(* IEC 61131-3 sources: Elmo_Master/test/Reports_Lasal/C78_20260806_preemption_cleanup_split (part 3) *)

		groupHeaderPublished := FALSE;
		if restorePreempt & restoredGroupActive then
			// The compact suffix is shared. Restore the complete captured suffix
			// even when the active Group is disjoint from the selected rollback
			// axes, and keep its shared header invalid until every record is done.
			identityHeaderBase := LMC_OWNER_IDENTITY_GROUP_HEADER_BASE;
			OwnershipIdentityState[identityHeaderBase] := 0;
			_memcpy(ptr1:=#OwnershipIdentityState[0],
				ptr2:=#OwnershipPreemptedIdentityState[0],
				cntr:=LMC_OWNER_IDENTITY_SUFFIX_BYTES);
			_memset(dest:=#OwnershipIdentityState[identityHeaderBase],
				usByte:=0, cntr:=40);
			OwnershipIdentityState[identityHeaderBase + 1] :=
				LMC_OWNER_IDENTITY_VERSION;
			OwnershipIdentityState[identityHeaderBase + 2]$UDINT :=
				restoredGroupIdentitySize;
			OwnershipIdentityState[identityHeaderBase + 3]$UDINT :=
				restoredGroupToken;
			OwnershipIdentityState[identityHeaderBase + 4]$UDINT :=
				restoredGroupGeneration;
			OwnershipIdentityState[identityHeaderBase + 5]$UDINT :=
				restoredGroupMask;
			OwnershipIdentityState[identityHeaderBase + 6]$UDINT :=
				restoredGroupSession;
			OwnershipIdentityState[identityHeaderBase + 7]$UDINT :=
				restoredGroupSequence;
			OwnershipIdentityState[identityHeaderBase + 8]$UDINT :=
				TO_UDINT(restoredGroupCommand) or
				(TO_UDINT(restoredGroupReference) shl 16);
			OwnershipIdentityState[identityHeaderBase + 9]$UDINT :=
				TO_UDINT(LMC_OWNER_KIND_GROUP) or
				(TO_UDINT(LMC_OWNER_RESOURCE_AXIS) shl 8) or
				(TO_UDINT(restoredGroupAdmissionMode) shl 16);
			groupHeaderPublished := TRUE;
		end_if;
		axisIndex := 1;
		while axisIndex <= LMC_OWNER_AXIS_COUNT do
			case axisIndex of
				1: axisBit := 0x00000001;
				2: axisBit := 0x00000002;
				3: axisBit := 0x00000004;
				4: axisBit := 0x00000008;
				5: axisBit := 0x00000010;
				6: axisBit := 0x00000020;
				7: axisBit := 0x00000040;
				8: axisBit := 0x00000080;
				9: axisBit := 0x00000100;
			else
				axisBit := 0;
			end_case;
			if (expectedAxisMask and axisBit) <> 0 then
				recordBase := LMC_OWNER_GLOBAL_SLOTS +
					((axisIndex - 1) * LMC_OWNER_AXIS_STRIDE);
				clearIndex := (axisIndex - 1) * LMC_OWNER_AXIS_STRIDE;
				observerBase := (axisIndex - 1) *
					LMC_OWNER_OBSERVER_STRIDE;
				identityHeaderBase := LMC_OWNER_IDENTITY_AXIS_HEADER_BASE +
					((axisIndex - 1) *
					 LMC_OWNER_IDENTITY_AXIS_HEADER_STRIDE);
				OwnershipIdentityState[identityHeaderBase] := 0;
				_memset(dest:=#OwnershipIdentityState[identityHeaderBase],
					usByte:=0,
					cntr:=LMC_OWNER_IDENTITY_AXIS_HEADER_STRIDE * 4);
				if restorePreempt then
					_memcpy(ptr1:=#OwnershipState[recordBase],
						ptr2:=#OwnershipPreemptedState[clearIndex],
						cntr:=LMC_OWNER_AXIS_STRIDE * 4);
					_memcpy(ptr1:=#OwnershipObserverState[observerBase],
						ptr2:=#OwnershipPreemptedIdentityState[
						 LMC_OWNER_PREEMPT_OBSERVER_BASE + observerBase],
						cntr:=LMC_OWNER_OBSERVER_STRIDE * 4);
				else
					_memcpy(ptr1:=#OwnershipState[recordBase],
						ptr2:=#OwnershipLeaseState[clearIndex],
						cntr:=LMC_OWNER_AXIS_STRIDE * 4);
					_memset(dest:=#OwnershipObserverState[observerBase],
						usByte:=0, cntr:=LMC_OWNER_OBSERVER_STRIDE * 4);
				end_if;
				if OwnershipState[recordBase + 1] <> LMC_OWNER_STATE_IDLE then
				identitySize := OwnershipState[recordBase + 15]$UDINT;
				identityTailSize := 0;
				if identitySize > LMC_OWNER_IDENTITY_PREFIX_BYTES then
					identityTailSize := identitySize -
						LMC_OWNER_IDENTITY_PREFIX_BYTES;
				end_if;
				identityPackedCommand :=
					TO_UDINT(OwnershipState[recordBase + 3]) or
					(TO_UDINT(OwnershipState[recordBase + 12]) shl 16);
				identityPackedOwner :=
					TO_UDINT(OwnershipState[recordBase + 2]) or
					(TO_UDINT(OwnershipState[recordBase + 13]) shl 8) or
					(TO_UDINT(OwnershipState[recordBase + 14]) shl 16);
				if OwnershipState[recordBase + 2] =
				   LMC_OWNER_KIND_GROUP then
					if groupHeaderPublished = FALSE then
						identityHeaderBase :=
							LMC_OWNER_IDENTITY_GROUP_HEADER_BASE;
						OwnershipIdentityState[identityHeaderBase] := 0;
						if restorePreempt then
							_memcpy(ptr1:=#OwnershipIdentityState[0],
								ptr2:=#OwnershipPreemptedIdentityState[0],
								cntr:=LMC_OWNER_IDENTITY_SUFFIX_BYTES);
							_memset(dest:=#OwnershipIdentityState[
								identityHeaderBase], usByte:=0, cntr:=40);
							OwnershipIdentityState[identityHeaderBase + 1] :=
								LMC_OWNER_IDENTITY_VERSION;
							OwnershipIdentityState[identityHeaderBase + 2]$UDINT :=
								identitySize;
							OwnershipIdentityState[identityHeaderBase + 3]$UDINT :=
								OwnershipState[recordBase + 4]$UDINT;
							OwnershipIdentityState[identityHeaderBase + 4]$UDINT :=
								OwnershipState[recordBase + 5]$UDINT;
							OwnershipIdentityState[identityHeaderBase + 5]$UDINT :=
								OwnershipState[recordBase + 11]$UDINT;
							OwnershipIdentityState[identityHeaderBase + 6]$UDINT :=
								OwnershipState[recordBase + 6]$UDINT;
							OwnershipIdentityState[identityHeaderBase + 7]$UDINT :=
								OwnershipState[recordBase + 7]$UDINT;
							OwnershipIdentityState[identityHeaderBase + 8]$UDINT :=
								identityPackedCommand;
							OwnershipIdentityState[identityHeaderBase + 9]$UDINT :=
								identityPackedOwner;
						else
							_memcpy(ptr1:=#OwnershipIdentityState[0],
								ptr2:=#OwnershipLeaseIdentityState[0],
								cntr:=LMC_OWNER_IDENTITY_SUFFIX_BYTES);
							_memset(dest:=#OwnershipIdentityState[
								identityHeaderBase], usByte:=0, cntr:=40);
							clearIndex := 1;
							while clearIndex <= 9 do
								OwnershipIdentityState[
									identityHeaderBase + clearIndex] :=
									OwnershipLeaseIdentityState[
									 LMC_OWNER_LEASE_IDENTITY_HEADER_BASE + clearIndex];
								clearIndex += 1;
							end_while;
						end_if;
						groupHeaderPublished := TRUE;
					end_if;
				else
					identityTailOffset :=
						TO_UDINT(OwnershipState[recordBase + 12] - 1) * 8;
					if restorePreempt then
						if identityTailSize > 0 then
							_memset(dest:=#OwnershipIdentityState[
								TO_DINT(identityTailOffset / 4)], usByte:=0,
								cntr:=identityTailSize);
							_memcpy(ptr1:=#OwnershipIdentityState[
								TO_DINT(identityTailOffset / 4)],
								ptr2:=#OwnershipPreemptedIdentityState[
								 TO_DINT(identityTailOffset / 4)],
								cntr:=identityTailSize);
						end_if;
					end_if;
					identityHeaderBase := LMC_OWNER_IDENTITY_AXIS_HEADER_BASE +
						((axisIndex - 1) *
						 LMC_OWNER_IDENTITY_AXIS_HEADER_STRIDE);
					OwnershipIdentityState[identityHeaderBase + 1] :=
						LMC_OWNER_IDENTITY_VERSION;
					OwnershipIdentityState[identityHeaderBase + 2]$UDINT :=
						identitySize;
					OwnershipIdentityState[identityHeaderBase + 3]$UDINT :=
						OwnershipState[recordBase + 4]$UDINT;
					OwnershipIdentityState[identityHeaderBase + 4]$UDINT :=
						OwnershipState[recordBase + 5]$UDINT;
					OwnershipIdentityState[identityHeaderBase + 5]$UDINT :=
						OwnershipState[recordBase + 11]$UDINT;
					OwnershipIdentityState[identityHeaderBase + 6]$UDINT :=
						OwnershipState[recordBase + 6]$UDINT;
					OwnershipIdentityState[identityHeaderBase + 7]$UDINT :=
						OwnershipState[recordBase + 7]$UDINT;
					OwnershipIdentityState[identityHeaderBase + 8]$UDINT :=
						identityPackedCommand;
					OwnershipIdentityState[identityHeaderBase + 9]$UDINT :=
						identityPackedOwner;
					OwnershipIdentityState[identityHeaderBase + 10]$UDINT :=
						identityTailOffset;
					OwnershipIdentityState[identityHeaderBase + 11]$UDINT :=
						identityTailSize;
					OwnershipIdentityState[identityHeaderBase]$UDINT :=
						LMC_OWNER_IDENTITY_AXIS_MAGIC + TO_UDINT(axisIndex);
				end_if;
				end_if;
			end_if;
			axisIndex += 1;
		end_while;
		if groupHeaderPublished then
			OwnershipIdentityState[
				LMC_OWNER_IDENTITY_GROUP_HEADER_BASE]$UDINT :=
				LMC_OWNER_IDENTITY_GROUP_MAGIC;
		end_if;

		if restorePreempt then
			OwnershipPreemptedIdentityState[
				LMC_OWNER_PREEMPT_HEADER_BASE] := 0;
			_memset(dest:=#OwnershipPreemptedState[0], usByte:=0,
				cntr:=sizeof(OwnershipPreemptedState));
			_memset(dest:=#OwnershipPreemptedIdentityState[0], usByte:=0,
				cntr:=sizeof(OwnershipPreemptedIdentityState));
			if restoredGroupActive = FALSE then
				OwnershipLeaseIdentityState[
					LMC_OWNER_LEASE_IDENTITY_HEADER_BASE] := 0;
				_memset(dest:=#OwnershipLeaseState[0], usByte:=0,
					cntr:=sizeof(OwnershipLeaseState));
				_memset(dest:=#OwnershipLeaseIdentityState[0], usByte:=0,
					cntr:=sizeof(OwnershipLeaseIdentityState));
			end_if;
		else
			OwnershipLeaseIdentityState[
				LMC_OWNER_LEASE_IDENTITY_HEADER_BASE] := 0;
			_memset(dest:=#OwnershipLeaseState[0], usByte:=0,
				cntr:=sizeof(OwnershipLeaseState));
			_memset(dest:=#OwnershipLeaseIdentityState[0], usByte:=0,
				cntr:=sizeof(OwnershipLeaseIdentityState));
		end_if;
	elsif Reason = 0 then
		axisIndex := 1;
		while axisIndex <= LMC_OWNER_AXIS_COUNT do
			case axisIndex of
				1: axisBit := 0x00000001;
				2: axisBit := 0x00000002;
				3: axisBit := 0x00000004;
				4: axisBit := 0x00000008;
				5: axisBit := 0x00000010;
				6: axisBit := 0x00000020;
				7: axisBit := 0x00000040;
				8: axisBit := 0x00000080;
				9: axisBit := 0x00000100;
			else
				axisBit := 0;
			end_case;
			if (expectedAxisMask and axisBit) <> 0 then
				recordBase := LMC_OWNER_GLOBAL_SLOTS +
					((axisIndex - 1) * LMC_OWNER_AXIS_STRIDE);
				observerBase := (axisIndex - 1) *
					LMC_OWNER_OBSERVER_STRIDE;
				identityHeaderBase := LMC_OWNER_IDENTITY_AXIS_HEADER_BASE +
					((axisIndex - 1) *
					 LMC_OWNER_IDENTITY_AXIS_HEADER_STRIDE);
				OwnershipIdentityState[identityHeaderBase] := 0;
				_memset(dest:=#OwnershipState[recordBase], usByte:=0,
					cntr:=LMC_OWNER_AXIS_STRIDE * 4);
				OwnershipState[recordBase] := axisIndex;
				OwnershipState[recordBase + 35]$UDINT :=
					LMC_OWNER_AXIS_RECORD_MAGIC + TO_UDINT(axisIndex);
				_memset(dest:=#OwnershipObserverState[observerBase], usByte:=0,
					cntr:=LMC_OWNER_OBSERVER_STRIDE * 4);
			end_if;
			axisIndex += 1;
		end_while;
		if expectedOwnerKind = LMC_OWNER_KIND_GROUP then
			OwnershipIdentityState[
				LMC_OWNER_IDENTITY_GROUP_HEADER_BASE] := 0;
			if expectedAdmissionMode <> LMC_OWNER_ADMISSION_SAFETY then
				_memset(dest:=#OwnershipIdentityState[0], usByte:=0,
					cntr:=LMC_OWNER_IDENTITY_SUFFIX_BYTES);
			end_if;
			_memset(dest:=#OwnershipIdentityState[
				LMC_OWNER_IDENTITY_GROUP_HEADER_BASE], usByte:=0, cntr:=40);
		elsif expectedIdentitySize > LMC_OWNER_IDENTITY_PREFIX_BYTES then
			identityTailSize := expectedIdentitySize -
				LMC_OWNER_IDENTITY_PREFIX_BYTES;
			identityTailOffset := TO_UDINT(expectedReference - 1) * 8;
			_memset(dest:=#OwnershipIdentityState[
				TO_DINT(identityTailOffset / 4)], usByte:=0,
				cntr:=identityTailSize);
		end_if;
	else
		axisIndex := 1;
		while axisIndex <= LMC_OWNER_AXIS_COUNT do
			case axisIndex of
				1: axisBit := 0x00000001;
				2: axisBit := 0x00000002;
				3: axisBit := 0x00000004;
				4: axisBit := 0x00000008;
				5: axisBit := 0x00000010;
				6: axisBit := 0x00000020;
				7: axisBit := 0x00000040;
				8: axisBit := 0x00000080;
				9: axisBit := 0x00000100;
			else
				axisBit := 0;
			end_case;
			if (expectedAxisMask and axisBit) <> 0 then
				recordBase := LMC_OWNER_GLOBAL_SLOTS +
					((axisIndex - 1) * LMC_OWNER_AXIS_STRIDE);
				OwnershipState[recordBase + 1] :=
					LMC_OWNER_STATE_QUARANTINED;
				OwnershipState[recordBase + 32] :=
					LMC_OWNER_REPORT_QUARANTINE;
				OwnershipState[recordBase + 33] := Reason;
			end_if;
			axisIndex += 1;
		end_while;
	end_if;
	if (Reason = 0) &
	   (OwnershipState[7]$UDINT = AdmissionToken) &
	   (OwnershipState[8]$UDINT = OwnerGeneration) then
		OwnershipState[7] := 0;
		OwnershipState[8] := 0;
		OwnershipState[9] := 0;
	end_if;
	if (Reason = 0) &
	   (OwnershipState[10]$UDINT = AdmissionToken) &
	   (OwnershipState[11]$UDINT = OwnerGeneration) then
		OwnershipState[10] := 0;
		OwnershipState[11] := 0;
		OwnershipState[12] := 0;
	end_if;
	if (Reason = 0) &
	   (OwnershipState[13]$UDINT = AdmissionToken) &
	   (OwnershipState[14]$UDINT = OwnerGeneration) then
		OwnershipState[13] := 0;
		OwnershipState[14] := 0;
		OwnershipState[15] := 0;
	end_if;
	Result := 0;

END_FUNCTION

FUNCTION GLOBAL LMCControlCommandService::PublishAxisOwnership
	VAR_INPUT
		AxisMask : UDINT;
		AdmissionToken : UDINT;
		OwnerGeneration : UDINT;
		ReportKind : UINT;
		ReportValue0 : UDINT;
		ReportValue1 : UDINT;
		ObservationCycle : UDINT;
	END_VAR
	VAR_OUTPUT
		Result : DINT;
	END_VAR
	VAR
		axisIndex : DINT;
		axisBit : UDINT;
		recordBase : DINT;
		firstRecordBase : DINT;
		leaseRecordBase : DINT;
		leaseFirstRecordBase : DINT;
		preemptRecordBase : DINT;
		probeRecordBase : DINT;
		probeAxisIndex : DINT;
		probeAxisBit : UDINT;
		observerBase : DINT;
		observerIndex : DINT;
		identityIndex : DINT;
		clearIndex : DINT;
		identityHeaderBase : DINT;
		identityCompareResult : UDINT;
		expectedResourceKind : DINT;
		expectedOwnerKind : DINT;
		expectedCommandId : DINT;
		expectedAdmissionMode : DINT;
		expectedReference : DINT;
		expectedSession : UDINT;
		expectedSequence : UDINT;
		observerFlags : UDINT;
		preemptFlags : UDINT;
		cleanupRequiredMask : UDINT;
		cleanupCompleteMask : UDINT;
		identitySize : UDINT;
		identityPrefixSize : UDINT;
		identityTailSize : UDINT;
		identityTailOffset : UDINT;
		identityPackedCommand : UDINT;
		identityPackedOwner : UDINT;
		preemptToken : UDINT;
		preemptGeneration : UDINT;
		preemptSession : UDINT;
		preemptSequence : UDINT;
		preemptMask : UDINT;
		preemptIdentitySize : UDINT;
		preemptState : DINT;
		preemptOwnerKind : DINT;
		preemptResourceKind : DINT;
		preemptCommand : DINT;
		preemptReference : DINT;
		preemptAdmission : DINT;
		replacementRecordBase : DINT;
		replacementHeaderBase : DINT;
		singletonToken : UDINT;
		singletonGeneration : UDINT;
		singletonMask : UDINT;
		replacementIdentitySize : UDINT;
		replacementTailSize : UDINT;
		replacementTailOffset : UDINT;
		replacementPackedCommand : UDINT;
		replacementPackedOwner : UDINT;
		resourceValid : BOOL;
		selectedFound : BOOL;
		identityShapeValid : BOOL;
		retainGroupLease : BOOL;
		forceQuarantine : BOOL;
		preemptRootValid : BOOL;
		cleanupReady : BOOL;
		restoreLease : BOOL;
		leaseValid : BOOL;
		retainLeaseValid : BOOL;
		preemptBankValid : BOOL;
		preemptSpecialValid : BOOL;
		replacementFound : BOOL;
		replacementValid : BOOL;
		replacementStateValid : BOOL;
		preemptLmcFound : BOOL;
		preemptDs402Found : BOOL;
		preemptEncoderFound : BOOL;
		destroyBanks : BOOL;
		clearOwner : BOOL;
		groupHeaderPublished : BOOL;
		homeReceiptExact : BOOL;
		homeReceiptCallMatches : BOOL;
		homeReceiptTerminalComplete : BOOL;
		homeReceiptAxisMaskValid : BOOL;
		homeReceiptIdentityPre : BOOL;
		homeReceiptIdentityPost : BOOL;
		homeReceiptObserverPre : BOOL;
		homeReceiptObserverPost : BOOL;
		homeReceiptRecordPre : BOOL;
		homeReceiptRecordBodyPost : BOOL;
		homeReceiptRecordPost : BOOL;
		homeReceiptSingletonPre : BOOL;
		homeReceiptSingletonPost : BOOL;
		homeReceiptSurfaceValid : BOOL;
		homeReceiptPhase : DINT;
		homeReceiptIndex : DINT;
		rebaseUpdateResult : DINT;
	END_VAR

	Result := -1;
	if (AxisMask = 0) | (AxisMask > LMC_OWNER_ROBOT_AXIS_MASK) |
	   (AdmissionToken = 0) | (OwnerGeneration = 0) |
	   (ReportKind < LMC_OWNER_REPORT_DISPATCH) |
	   (ReportKind > LMC_OWNER_REPORT_SAFETY_PREEMPT) then
		RETURN;
	end_if;
	if ZeroHomeState[60]$UDINT = LMC_HOME_OWNER_RECEIPT_MAGIC then
		homeReceiptCallMatches :=
			(ZeroHomeState[34]$UDINT = AdmissionToken) &
			(ZeroHomeState[35]$UDINT = OwnerGeneration) &
			(ZeroHomeState[38]$UDINT = AxisMask) &
			(ZeroHomeState[58] = TO_DINT(ReportKind)) &
			(ZeroHomeState[57]$UDINT = ReportValue0) &
			(ZeroHomeState[31]$UDINT = ReportValue1) &
			(ZeroHomeState[46]$UDINT = ObservationCycle);
		homeReceiptTerminalComplete :=
			(ZeroHomeState[51]$UDINT = LMC_HOME_RECORD_MAGIC) &
			(ZeroHomeState[33]$UDINT <> 0) &
			(ZeroHomeState[63]$UDINT = ZeroHomeState[33]$UDINT) &
			(ZeroHomeState[62] = 0) &
			(ZeroHomeState[61] = LMC_HOME_OWNER_RECEIPT_COMPLETE) &
			(ZeroHomeState[59] = 0) &
			(ZeroHomeState[39] = LMC_HOME_ENGINE_TERMINAL) &
			(ZeroHomeState[0] >= LMC_HOME_RECORD_SUCCEEDED) &
			(ZeroHomeState[0] <= LMC_HOME_RECORD_ABORTED) &
			(ZeroHomeState[57] = ZeroHomeState[0]) &
			(ZeroHomeState[47] = 1) &
			((ZeroHomeState[56]$UDINT and
			  LMC_HOME_FLAG_OWNER_FINALIZE_ACCEPTED) <> 0) &
			((ZeroHomeState[56]$UDINT and
			  LMC_HOME_FLAG_TERMINAL_PUBLISHED) <> 0) &
			((ZeroHomeState[56]$UDINT and
			  LMC_HOME_FLAG_PREEMPTION_CLEANUP) = 0) &
			(((ZeroHomeState[0] = LMC_HOME_RECORD_SUCCEEDED) &
			  (ZeroHomeState[58] = LMC_OWNER_REPORT_TERMINAL_SUCCESS)) |
			 (((ZeroHomeState[0] = LMC_HOME_RECORD_FAILED) |
			   (ZeroHomeState[0] = LMC_HOME_RECORD_ABORTED)) &
			  (ZeroHomeState[58] =
			   LMC_OWNER_REPORT_TERMINAL_SAFE_FAILURE)));
		if homeReceiptCallMatches then
		homeReceiptPhase := ZeroHomeState[61];
		homeReceiptAxisMaskValid := FALSE;
		case ZeroHomeState[9] of
			1: homeReceiptAxisMaskValid := AxisMask = 0x00000001;
			2: homeReceiptAxisMaskValid := AxisMask = 0x00000002;
			3: homeReceiptAxisMaskValid := AxisMask = 0x00000004;
			4: homeReceiptAxisMaskValid := AxisMask = 0x00000008;
		else
		end_case;
		homeReceiptExact :=
			homeReceiptAxisMaskValid &
			(ZeroHomeState[51]$UDINT = LMC_HOME_RECORD_MAGIC) &
			(ZeroHomeState[33]$UDINT <> 0) &
			(ZeroHomeState[63]$UDINT = ZeroHomeState[33]$UDINT) &
			(ZeroHomeState[62] = 0) &
			(ZeroHomeState[34]$UDINT = AdmissionToken) &
			(ZeroHomeState[35]$UDINT = OwnerGeneration) &
			(ZeroHomeState[38]$UDINT = AxisMask) &
			(ZeroHomeState[58] = TO_DINT(ReportKind)) &
			(ZeroHomeState[57]$UDINT = ReportValue0) &
			(ZeroHomeState[31]$UDINT = ReportValue1) &
			(ZeroHomeState[46]$UDINT = ObservationCycle) &
			(ZeroHomeState[59] = 0) &
			((ZeroHomeState[39] = LMC_HOME_ENGINE_FINALIZE) |
			 (ZeroHomeState[39] = LMC_HOME_ENGINE_TERMINAL)) &
			((ZeroHomeState[56]$UDINT and
			  LMC_HOME_FLAG_OWNER_FINALIZE_INTENT) <> 0) &
			((ZeroHomeState[56]$UDINT and
			  LMC_HOME_FLAG_PREEMPTION_CLEANUP) = 0) &
			((ReportKind = LMC_OWNER_REPORT_TERMINAL_SUCCESS) |
			 (ReportKind = LMC_OWNER_REPORT_TERMINAL_SAFE_FAILURE)) &
			(homeReceiptPhase >= LMC_HOME_OWNER_RECEIPT_PREPARED) &
			(homeReceiptPhase <= LMC_HOME_OWNER_RECEIPT_COMPLETE);
		if homeReceiptExact = FALSE then
			OwnershipState[24] := 1;
			Result := -3;
			RETURN;
		end_if;

		axisIndex := ZeroHomeState[9];
		recordBase := LMC_OWNER_GLOBAL_SLOTS +
			((axisIndex - 1) * LMC_OWNER_AXIS_STRIDE);
		observerBase := (axisIndex - 1) * LMC_OWNER_OBSERVER_STRIDE;
		identityHeaderBase := LMC_OWNER_IDENTITY_AXIS_HEADER_BASE +
			((axisIndex - 1) * LMC_OWNER_IDENTITY_AXIS_HEADER_STRIDE);
		identityPackedCommand := TO_UDINT(0x7D13) or
			(TO_UDINT(axisIndex) shl 16);
		identityPackedOwner := TO_UDINT(LMC_OWNER_KIND_LMC_HOME) or
			(TO_UDINT(LMC_OWNER_RESOURCE_LMC_HOME_ENGINE) shl 8) or
			(TO_UDINT(LMC_OWNER_ADMISSION_LIFECYCLE) shl 16);
		identitySize := OwnershipState[recordBase + 15]$UDINT;
		identityTailOffset := TO_UDINT(axisIndex - 1) * 8;
		identityTailSize := 0;
		if identitySize > LMC_OWNER_IDENTITY_PREFIX_BYTES then
			identityTailSize := identitySize - LMC_OWNER_IDENTITY_PREFIX_BYTES;
		end_if;

		homeReceiptIdentityPre :=
			(OwnershipIdentityState[identityHeaderBase]$UDINT =
			 (LMC_OWNER_IDENTITY_AXIS_MAGIC + TO_UDINT(axisIndex))) &
			(OwnershipIdentityState[identityHeaderBase + 1] =
			 LMC_OWNER_IDENTITY_VERSION) &
			(OwnershipIdentityState[identityHeaderBase + 2]$UDINT = 56) &
			(OwnershipIdentityState[identityHeaderBase + 3]$UDINT =
			 AdmissionToken) &
			(OwnershipIdentityState[identityHeaderBase + 4]$UDINT =
			 OwnerGeneration) &
			(OwnershipIdentityState[identityHeaderBase + 5]$UDINT = AxisMask) &
			(OwnershipIdentityState[identityHeaderBase + 6]$UDINT =
			 ZeroHomeState[36]$UDINT) &
			(OwnershipIdentityState[identityHeaderBase + 7]$UDINT =
			 ZeroHomeState[37]$UDINT) &
			(OwnershipIdentityState[identityHeaderBase + 8]$UDINT =
			 identityPackedCommand) &
			(OwnershipIdentityState[identityHeaderBase + 9]$UDINT =
			 identityPackedOwner) &
			(OwnershipIdentityState[identityHeaderBase + 10]$UDINT =
			 identityTailOffset) &
			(OwnershipIdentityState[identityHeaderBase + 11]$UDINT = 0) &
			(identitySize = 56) & (identityTailSize = 0);
		homeReceiptIdentityPost := TRUE;
		homeReceiptIndex := 0;
		while homeReceiptIndex < LMC_OWNER_IDENTITY_AXIS_HEADER_STRIDE do
			if OwnershipIdentityState[identityHeaderBase + homeReceiptIndex] <> 0 then
				homeReceiptIdentityPost := FALSE;
			end_if;
			homeReceiptIndex += 1;
		end_while;

		homeReceiptObserverPre :=
			(OwnershipObserverState[observerBase]$UDINT =
			 (LMC_OWNER_OBSERVER_MAGIC + TO_UDINT(axisIndex))) &
			(OwnershipObserverState[observerBase + 1]$UDINT = AdmissionToken) &
			(OwnershipObserverState[observerBase + 2]$UDINT = OwnerGeneration) &
			((OwnershipObserverState[observerBase + 5]$UDINT and
			  LMC_OWNER_OBSERVER_EVIDENCE_CLEAR_MASK) = 0) &
			(OwnershipObserverState[observerBase + 9] = 0) &
			(OwnershipObserverState[observerBase + 10] = 0) &
			(OwnershipObserverState[observerBase + 11] = 0);
		homeReceiptObserverPost := TRUE;
		homeReceiptIndex := 0;
		while homeReceiptIndex < LMC_OWNER_OBSERVER_STRIDE do
			if OwnershipObserverState[observerBase + homeReceiptIndex] <> 0 then
				homeReceiptObserverPost := FALSE;
			end_if;
			homeReceiptIndex += 1;
		end_while;

		homeReceiptRecordPre :=
			(OwnershipState[recordBase] = axisIndex) &
			(OwnershipState[recordBase + 1] = LMC_OWNER_STATE_LMC_HOME_ACTIVE) &
			(OwnershipState[recordBase + 2] = LMC_OWNER_KIND_LMC_HOME) &
			(OwnershipState[recordBase + 3] = 0x7D13) &
			(OwnershipState[recordBase + 4]$UDINT = AdmissionToken) &
			(OwnershipState[recordBase + 5]$UDINT = OwnerGeneration) &
			(OwnershipState[recordBase + 6]$UDINT = ZeroHomeState[36]$UDINT) &
			(OwnershipState[recordBase + 7]$UDINT = ZeroHomeState[37]$UDINT) &
			(OwnershipState[recordBase + 8]$UDINT <> 0) &
			(OwnershipState[recordBase + 9]$UDINT <> 0) &
			(OwnershipState[recordBase + 10] = 0) &
			(OwnershipState[recordBase + 11]$UDINT = AxisMask) &
			(OwnershipState[recordBase + 12] = axisIndex) &
			(OwnershipState[recordBase + 13] =
			 LMC_OWNER_RESOURCE_LMC_HOME_ENGINE) &
			(OwnershipState[recordBase + 14] =
			 LMC_OWNER_ADMISSION_LIFECYCLE) &
			(OwnershipState[recordBase + 15]$UDINT = 56) &
			(OwnershipState[recordBase + 16]$UDINT = 1) &
			(OwnershipState[recordBase + 17]$UDINT = ZeroHomeState[4]$UDINT) &
			(OwnershipState[recordBase + 18]$UDINT = ZeroHomeState[1]$UDINT) &
			(OwnershipState[recordBase + 19]$UDINT = ZeroHomeState[2]$UDINT) &
			(OwnershipState[recordBase + 20]$UDINT = ZeroHomeState[3]$UDINT) &
			(OwnershipState[recordBase + 21]$UDINT = ZeroHomeState[5]$UDINT) &
			(OwnershipState[recordBase + 22]$UDINT = ZeroHomeState[6]$UDINT) &
			(OwnershipState[recordBase + 23]$UDINT = ZeroHomeState[7]$UDINT) &
			(OwnershipState[recordBase + 24]$UDINT = ZeroHomeState[8]$UDINT) &
			(OwnershipState[recordBase + 25]$UDINT = 1) &
			(OwnershipState[recordBase + 26] = ZeroHomeState[11]) &
			(OwnershipState[recordBase + 27] = ZeroHomeState[12]) &
			(OwnershipState[recordBase + 28]$UDINT = ZeroHomeState[13]$UDINT) &
			(OwnershipState[recordBase + 29]$UDINT = 0x454D4F48) &
			(OwnershipState[recordBase + 30] = 0) &
			(OwnershipState[recordBase + 31] = 0) &
			(OwnershipState[recordBase + 32] = 0) &
			(OwnershipState[recordBase + 33] = 0) &
			(OwnershipState[recordBase + 34] = 0) &
			(OwnershipState[recordBase + 35]$UDINT =
			 (LMC_OWNER_AXIS_RECORD_MAGIC + TO_UDINT(axisIndex)));
		homeReceiptRecordBodyPost := OwnershipState[recordBase] = axisIndex;
		homeReceiptIndex := 1;
		while homeReceiptIndex <= 34 do
			if OwnershipState[recordBase + homeReceiptIndex] <> 0 then
				homeReceiptRecordBodyPost := FALSE;
			end_if;
			homeReceiptIndex += 1;
		end_while;
		homeReceiptRecordPost := homeReceiptRecordBodyPost &
			(OwnershipState[recordBase + 35]$UDINT =
			 (LMC_OWNER_AXIS_RECORD_MAGIC + TO_UDINT(axisIndex)));
		homeReceiptSingletonPre :=
			(OwnershipState[7]$UDINT = AdmissionToken) &
			(OwnershipState[8]$UDINT = OwnerGeneration) &
			(OwnershipState[9]$UDINT = AxisMask);
		homeReceiptSingletonPost :=
			(OwnershipState[7]$UDINT = 0) &
			(OwnershipState[8]$UDINT = 0) &
			(OwnershipState[9]$UDINT = 0);

		homeReceiptSurfaceValid := FALSE;
		case homeReceiptPhase of
			LMC_HOME_OWNER_RECEIPT_PREPARED:
				homeReceiptSurfaceValid := homeReceiptIdentityPre &
					homeReceiptObserverPre & homeReceiptRecordPre &
					homeReceiptSingletonPre;
			LMC_HOME_OWNER_RECEIPT_CLEAR_IDENTITY:
				homeReceiptSurfaceValid :=
					(homeReceiptIdentityPre | homeReceiptIdentityPost |
					 (OwnershipIdentityState[identityHeaderBase] = 0)) &
					homeReceiptObserverPre & homeReceiptRecordPre &
					homeReceiptSingletonPre;
			LMC_HOME_OWNER_RECEIPT_CLEAR_OBSERVER:
				homeReceiptSurfaceValid := homeReceiptIdentityPost &
					(homeReceiptObserverPre | homeReceiptObserverPost |
					 (OwnershipObserverState[observerBase] = 0)) &
					homeReceiptRecordPre & homeReceiptSingletonPre;
			LMC_HOME_OWNER_RECEIPT_CLEAR_SINGLETON:
				homeReceiptSurfaceValid := homeReceiptIdentityPost &
					homeReceiptObserverPost & homeReceiptRecordPre &
					(homeReceiptSingletonPre |
					 ((OwnershipState[7]$UDINT = 0) &
					  (OwnershipState[8]$UDINT = OwnerGeneration) &
					  (OwnershipState[9]$UDINT = AxisMask)) |
					 ((OwnershipState[7]$UDINT = 0) &
					  (OwnershipState[8]$UDINT = 0) &
					  (OwnershipState[9]$UDINT = AxisMask)) |
					 homeReceiptSingletonPost);
			LMC_HOME_OWNER_RECEIPT_CLEAR_RECORD:
				homeReceiptSurfaceValid := homeReceiptIdentityPost &
					homeReceiptObserverPost & homeReceiptSingletonPost &
					(homeReceiptRecordPre |
					 (OwnershipState[recordBase + 35] = 0));
			LMC_HOME_OWNER_RECEIPT_COMPLETE:
				homeReceiptSurfaceValid := homeReceiptIdentityPost &
					homeReceiptObserverPost & homeReceiptSingletonPost &
					(homeReceiptRecordPost |
					 (homeReceiptRecordBodyPost &
					  (OwnershipState[recordBase + 35] = 0)));
		else
		end_case;
		if homeReceiptSurfaceValid = FALSE then
			OwnershipState[24] := 1;
			Result := -3;
			RETURN;
		end_if;
		if (ZeroHomeState[56]$UDINT and
		   LMC_HOME_FLAG_OWNER_FINALIZE_ACCEPTED) = 0 then
			if homeReceiptPhase <> LMC_HOME_OWNER_RECEIPT_PREPARED then
				OwnershipState[24] := 1;
				Result := -3;
				RETURN;
			end_if;
			Result := 0;
			RETURN;
		end_if;

		// The axis-record magic is committed last. Each phase is stored before its
		// mutation, so the exact receipt can resume a partial cleanup fail-closed.
		if homeReceiptPhase <= LMC_HOME_OWNER_RECEIPT_CLEAR_IDENTITY then
			ZeroHomeState[61] := LMC_HOME_OWNER_RECEIPT_CLEAR_IDENTITY;
			OwnershipIdentityState[identityHeaderBase] := 0;
			_memset(dest:=#OwnershipIdentityState[identityHeaderBase],
				usByte:=0, cntr:=LMC_OWNER_IDENTITY_AXIS_HEADER_STRIDE * 4);
		end_if;
		if homeReceiptPhase <= LMC_HOME_OWNER_RECEIPT_CLEAR_OBSERVER then
			ZeroHomeState[61] := LMC_HOME_OWNER_RECEIPT_CLEAR_OBSERVER;
			OwnershipObserverState[observerBase] := 0;
			_memset(dest:=#OwnershipObserverState[observerBase],
				usByte:=0, cntr:=LMC_OWNER_OBSERVER_STRIDE * 4);
		end_if;
		if homeReceiptPhase <= LMC_HOME_OWNER_RECEIPT_CLEAR_SINGLETON then
			ZeroHomeState[61] := LMC_HOME_OWNER_RECEIPT_CLEAR_SINGLETON;
			OwnershipState[7] := 0;
			OwnershipState[8] := 0;
			OwnershipState[9] := 0;
		end_if;
		if homeReceiptPhase <= LMC_HOME_OWNER_RECEIPT_CLEAR_RECORD then
			ZeroHomeState[61] := LMC_HOME_OWNER_RECEIPT_CLEAR_RECORD;
			OwnershipState[recordBase + 35] := 0;
			_memset(dest:=#OwnershipState[recordBase], usByte:=0,
				cntr:=LMC_OWNER_AXIS_STRIDE * 4);
			OwnershipState[recordBase] := axisIndex;
			ZeroHomeState[61] := LMC_HOME_OWNER_RECEIPT_COMPLETE;
			OwnershipState[recordBase + 35]$UDINT :=
				LMC_OWNER_AXIS_RECORD_MAGIC + TO_UDINT(axisIndex);
		elsif (homeReceiptPhase = LMC_HOME_OWNER_RECEIPT_COMPLETE) &
		      homeReceiptRecordBodyPost &
		      (OwnershipState[recordBase + 35] = 0) then
			OwnershipState[recordBase + 35]$UDINT :=
				LMC_OWNER_AXIS_RECORD_MAGIC + TO_UDINT(axisIndex);
		end_if;
		if (ZeroHomeState[61] <> LMC_HOME_OWNER_RECEIPT_COMPLETE) |
		   (OwnershipState[recordBase + 35]$UDINT <>
		    (LMC_OWNER_AXIS_RECORD_MAGIC + TO_UDINT(axisIndex))) then
			OwnershipState[24] := 1;
			Result := -3;
			RETURN;
		end_if;
		// Clear only after exact successful Home and durable owner cleanup. The
		// caller has not published ZeroHomeState[0] yet, so the receipt-bound
		// terminal tuple is the authoritative success proof at this point.
		if LMC_AXIS_REBASE_BARRIER_ENABLED &
		   (ReportKind = LMC_OWNER_REPORT_TERMINAL_SUCCESS) &
		   (ReportValue0 = LMC_HOME_RECORD_SUCCEEDED) &
		   (ZeroHomeState[57] = LMC_HOME_RECORD_SUCCEEDED) then
			rebaseUpdateResult := UpdateAxisRebaseRequiredState(
				SetAxisMask:=0, ClearAxisMask:=AxisMask);
			if rebaseUpdateResult <> 0 then
				Result := rebaseUpdateResult;
				RETURN;
			end_if;
		end_if;
		Result := 1;
		RETURN;
		elsif homeReceiptTerminalComplete = FALSE then
			OwnershipState[24] := 1;
			Result := -3;
			RETURN;
		end_if;
	end_if;
	expectedResourceKind := 0;
	expectedOwnerKind := 0;
	expectedCommandId := 0;
	expectedAdmissionMode := 0;
	expectedReference := 0;
	expectedSession := 0;
	expectedSequence := 0;
	identitySize := 0;
	firstRecordBase := -1;
	selectedFound := FALSE;
	axisIndex := 1;
	while axisIndex <= LMC_OWNER_AXIS_COUNT do
		case axisIndex of
			1: axisBit := 0x00000001;
			2: axisBit := 0x00000002;
			3: axisBit := 0x00000004;
			4: axisBit := 0x00000008;
			5: axisBit := 0x00000010;
			6: axisBit := 0x00000020;
			7: axisBit := 0x00000040;
			8: axisBit := 0x00000080;
			9: axisBit := 0x00000100;
		else
			axisBit := 0;
		end_case;
		recordBase := LMC_OWNER_GLOBAL_SLOTS +
			((axisIndex - 1) * LMC_OWNER_AXIS_STRIDE);
		if (AxisMask and axisBit) <> 0 then
			if selectedFound = FALSE then
				expectedResourceKind := OwnershipState[recordBase + 13];
				expectedOwnerKind := OwnershipState[recordBase + 2];
				expectedCommandId := OwnershipState[recordBase + 3];
				expectedAdmissionMode := OwnershipState[recordBase + 14];
				expectedReference := OwnershipState[recordBase + 12];
				expectedSession := OwnershipState[recordBase + 6]$UDINT;
				expectedSequence := OwnershipState[recordBase + 7]$UDINT;
				identitySize := OwnershipState[recordBase + 15]$UDINT;
				firstRecordBase := recordBase;
				selectedFound := TRUE;
			end_if;
			if (OwnershipState[recordBase] <> axisIndex) |
			   (OwnershipState[recordBase + 35]$UDINT <>
			    (LMC_OWNER_AXIS_RECORD_MAGIC + TO_UDINT(axisIndex))) |
			   (OwnershipState[recordBase + 4]$UDINT <>
			    AdmissionToken) |
			   (OwnershipState[recordBase + 5]$UDINT <>
			    OwnerGeneration) |
			   (OwnershipState[recordBase + 11]$UDINT <> AxisMask) |
			   (OwnershipState[recordBase + 13] <>
			    expectedResourceKind) |
			   (OwnershipState[recordBase + 2] <> expectedOwnerKind) |
			   (OwnershipState[recordBase + 3] <> expectedCommandId) |
			   (OwnershipState[recordBase + 14] <>
			    expectedAdmissionMode) |
			   (OwnershipState[recordBase + 12] <>
			    expectedReference) |
			   (OwnershipState[recordBase + 6]$UDINT <> expectedSession) |
			   (OwnershipState[recordBase + 7]$UDINT <> expectedSequence) |
			   (OwnershipState[recordBase + 15]$UDINT <> identitySize) then
				Result := -2;
				RETURN;
			elsif (OwnershipState[recordBase + 1] =
			       LMC_OWNER_STATE_QUARANTINED) &
			      (ReportKind <> LMC_OWNER_REPORT_QUARANTINE) then
				Result := -3;
				RETURN;
			end_if;
		elsif (OwnershipState[recordBase + 4]$UDINT = AdmissionToken) |
		      (OwnershipState[recordBase + 5]$UDINT = OwnerGeneration) then
			Result := -2;
			RETURN;
		end_if;
		axisIndex += 1;
	end_while;
	if selectedFound = FALSE then
		Result := -2;
		RETURN;
	end_if;
	identityShapeValid := FALSE;
	if expectedCommandId = 0x2023 then
		identityShapeValid := identitySize = 8;
	elsif expectedCommandId = 0x2024 then
		identityShapeValid := identitySize = 1;
	elsif expectedCommandId = 0x2022 then
		identityShapeValid := identitySize = 16;
	elsif (expectedCommandId = 0x209F) | (expectedCommandId = 0x20A0) then
		identityShapeValid := identitySize = 32;
	elsif expectedCommandId = 0x20A2 then
		identityShapeValid := identitySize = 24;
	elsif (expectedCommandId = 0x2047) | (expectedCommandId = 0x2048) |
	      (expectedCommandId = 0x2049) | (expectedCommandId = 0x204A) |
	      (expectedCommandId = 0x204B) then
		identityShapeValid := identitySize = 1;
	elsif expectedCommandId = 0x2085 then
		identityShapeValid := identitySize = 16;
	elsif expectedCommandId = 0x20A4 then
		identityShapeValid := identitySize = 96;
	elsif expectedCommandId = 0x7D22 then
		identityShapeValid := identitySize = 104;
	elsif expectedCommandId = 0x20E7 then
		identityShapeValid := identitySize = 1320;
	elsif expectedCommandId = 0x7D13 then
		identityShapeValid := identitySize = 56;
	elsif (expectedCommandId = 0x7D15) |
	      (expectedCommandId = 0x7E53) then
		identityShapeValid := identitySize = 72;
	end_if;
	identityPrefixSize := identitySize;
	if identityPrefixSize > LMC_OWNER_IDENTITY_PREFIX_BYTES then
		identityPrefixSize := LMC_OWNER_IDENTITY_PREFIX_BYTES;
	end_if;
	identityTailSize := 0;
	if identitySize > LMC_OWNER_IDENTITY_PREFIX_BYTES then
		identityTailSize := identitySize - LMC_OWNER_IDENTITY_PREFIX_BYTES;
	end_if;
	identityTailOffset := 0;
	if expectedOwnerKind <> LMC_OWNER_KIND_GROUP then
		if (expectedReference < 1) |
		   (expectedReference > LMC_OWNER_AXIS_COUNT) then
			identityShapeValid := FALSE;
		else
			identityTailOffset := TO_UDINT(expectedReference - 1) * 8;
		end_if;
		if identityTailSize > 8 then
			identityShapeValid := FALSE;
		end_if;
	end_if;
	if (identityTailOffset + identityTailSize) >
	   LMC_OWNER_IDENTITY_SUFFIX_BYTES then
		identityShapeValid := FALSE;
	end_if;
	identityPackedCommand := TO_UDINT(expectedCommandId) or
		(TO_UDINT(expectedReference) shl 16);
	identityPackedOwner := TO_UDINT(expectedOwnerKind) or
		(TO_UDINT(expectedResourceKind) shl 8) or
		(TO_UDINT(expectedAdmissionMode) shl 16);
	axisIndex := 1;
	while axisIndex <= LMC_OWNER_AXIS_COUNT do
		case axisIndex of
			1: axisBit := 0x00000001;
			2: axisBit := 0x00000002;
			3: axisBit := 0x00000004;
			4: axisBit := 0x00000008;
			5: axisBit := 0x00000010;
			6: axisBit := 0x00000020;
			7: axisBit := 0x00000040;
			8: axisBit := 0x00000080;
			9: axisBit := 0x00000100;
		else
			axisBit := 0;
		end_case;
		if (AxisMask and axisBit) <> 0 then
			recordBase := LMC_OWNER_GLOBAL_SLOTS +
				((axisIndex - 1) * LMC_OWNER_AXIS_STRIDE);
			if expectedOwnerKind = LMC_OWNER_KIND_GROUP then
				identityHeaderBase := LMC_OWNER_IDENTITY_GROUP_HEADER_BASE;
				if (OwnershipIdentityState[identityHeaderBase]$UDINT <>
				    LMC_OWNER_IDENTITY_GROUP_MAGIC) |
				   (OwnershipIdentityState[identityHeaderBase + 1] <>
				    LMC_OWNER_IDENTITY_VERSION) |
				   (OwnershipIdentityState[identityHeaderBase + 2]$UDINT <>
				    identitySize) |
				   (OwnershipIdentityState[identityHeaderBase + 3]$UDINT <>
				    AdmissionToken) |
				   (OwnershipIdentityState[identityHeaderBase + 4]$UDINT <>
				    OwnerGeneration) |
				   (OwnershipIdentityState[identityHeaderBase + 5]$UDINT <>
				    AxisMask) |
				   (OwnershipIdentityState[identityHeaderBase + 6]$UDINT <>
				    expectedSession) |
				   (OwnershipIdentityState[identityHeaderBase + 7]$UDINT <>
				    expectedSequence) |
				   (OwnershipIdentityState[identityHeaderBase + 8]$UDINT <>
				    identityPackedCommand) |
				   (OwnershipIdentityState[identityHeaderBase + 9]$UDINT <>
				    identityPackedOwner) then
					identityShapeValid := FALSE;
				end_if;
			else
				identityHeaderBase := LMC_OWNER_IDENTITY_AXIS_HEADER_BASE +
					((axisIndex - 1) * LMC_OWNER_IDENTITY_AXIS_HEADER_STRIDE);
				if (OwnershipIdentityState[identityHeaderBase]$UDINT <>
				    (LMC_OWNER_IDENTITY_AXIS_MAGIC + TO_UDINT(axisIndex))) |
				   (OwnershipIdentityState[identityHeaderBase + 1] <>
				    LMC_OWNER_IDENTITY_VERSION) |
				   (OwnershipIdentityState[identityHeaderBase + 2]$UDINT <>
				    identitySize) |
				   (OwnershipIdentityState[identityHeaderBase + 3]$UDINT <>
				    AdmissionToken) |
				   (OwnershipIdentityState[identityHeaderBase + 4]$UDINT <>
				    OwnerGeneration) |
				   (OwnershipIdentityState[identityHeaderBase + 5]$UDINT <>
				    AxisMask) |
				   (OwnershipIdentityState[identityHeaderBase + 6]$UDINT <>
				    expectedSession) |
				   (OwnershipIdentityState[identityHeaderBase + 7]$UDINT <>
				    expectedSequence) |
				   (OwnershipIdentityState[identityHeaderBase + 8]$UDINT <>
				    identityPackedCommand) |
				   (OwnershipIdentityState[identityHeaderBase + 9]$UDINT <>
				    identityPackedOwner) |
				   (OwnershipIdentityState[identityHeaderBase + 10]$UDINT <>
				    identityTailOffset) |
				   (OwnershipIdentityState[identityHeaderBase + 11]$UDINT <>
				    identityTailSize) then
					identityShapeValid := FALSE;
				end_if;
			end_if;
			identityCompareResult := _memcmp(
				ptr1:=#OwnershipState[firstRecordBase + 16],
				ptr2:=#OwnershipState[recordBase + 16],
				cntr:=identityPrefixSize);
			if identityCompareResult <> 0 then
				identityShapeValid := FALSE;
			end_if;
		end_if;
		axisIndex += 1;
	end_while;
	if identityShapeValid = FALSE then
		OwnershipState[24] := 1;
		Result := -3;
		RETURN;
	end_if;
	resourceValid := FALSE;
	case expectedResourceKind of
		LMC_OWNER_RESOURCE_AXIS:
			resourceValid :=
				(OwnershipState[7]$UDINT <> AdmissionToken) &
				(OwnershipState[8]$UDINT <> OwnerGeneration) &
				(OwnershipState[10]$UDINT <> AdmissionToken) &
				(OwnershipState[11]$UDINT <> OwnerGeneration) &
				(OwnershipState[13]$UDINT <> AdmissionToken) &
				(OwnershipState[14]$UDINT <> OwnerGeneration);
		LMC_OWNER_RESOURCE_LMC_HOME_ENGINE:
			resourceValid :=
				(OwnershipState[7]$UDINT = AdmissionToken) &
				(OwnershipState[8]$UDINT = OwnerGeneration) &
				(OwnershipState[9]$UDINT = AxisMask) &
				(OwnershipState[10]$UDINT <> AdmissionToken) &
				(OwnershipState[11]$UDINT <> OwnerGeneration) &
				(OwnershipState[13]$UDINT <> AdmissionToken) &
				(OwnershipState[14]$UDINT <> OwnerGeneration);
		LMC_OWNER_RESOURCE_DS402_HOME_ENGINE:
			resourceValid :=
				(OwnershipState[10]$UDINT = AdmissionToken) &
				(OwnershipState[11]$UDINT = OwnerGeneration) &
				(OwnershipState[12]$UDINT = AxisMask) &
				(OwnershipState[7]$UDINT <> AdmissionToken) &
				(OwnershipState[8]$UDINT <> OwnerGeneration) &
				(OwnershipState[13]$UDINT <> AdmissionToken) &
				(OwnershipState[14]$UDINT <> OwnerGeneration);
		LMC_OWNER_RESOURCE_DIAGNOSTICS_SDO_ENGINE:
			resourceValid :=
				(OwnershipState[13]$UDINT = AdmissionToken) &
				(OwnershipState[14]$UDINT = OwnerGeneration) &
				(OwnershipState[15]$UDINT = AxisMask) &
				(OwnershipState[7]$UDINT <> AdmissionToken) &
				(OwnershipState[8]$UDINT <> OwnerGeneration) &
				(OwnershipState[10]$UDINT <> AdmissionToken) &
				(OwnershipState[11]$UDINT <> OwnerGeneration);
	else
	end_case;
	if resourceValid = FALSE then
		Result := -2;
		RETURN;
	end_if;

	preemptRootValid :=
		(OwnershipPreemptedIdentityState[
		 LMC_OWNER_PREEMPT_HEADER_BASE]$UDINT =
		 LMC_OWNER_PREEMPT_IDENTITY_MAGIC) &
		(OwnershipPreemptedIdentityState[
		 LMC_OWNER_PREEMPT_HEADER_BASE + 2]$UDINT = AdmissionToken) &
		(OwnershipPreemptedIdentityState[
		 LMC_OWNER_PREEMPT_HEADER_BASE + 3]$UDINT = OwnerGeneration) &
		(OwnershipPreemptedIdentityState[
		 LMC_OWNER_PREEMPT_HEADER_BASE + 4]$UDINT = AxisMask) &
		(OwnershipPreemptedIdentityState[
		 LMC_OWNER_PREEMPT_HEADER_BASE + 5]$UDINT = expectedSession) &
		(OwnershipPreemptedIdentityState[
		 LMC_OWNER_PREEMPT_HEADER_BASE + 6]$UDINT = expectedSequence) &
		(OwnershipPreemptedIdentityState[
		 LMC_OWNER_PREEMPT_HEADER_BASE + 7]$UDINT =
		 (TO_UDINT(expectedCommandId) or
		  (TO_UDINT(expectedReference) shl 16))) &
		((OwnershipPreemptedIdentityState[
		  LMC_OWNER_PREEMPT_HEADER_BASE + 1]$UDINT and 0x0000FFFF) =
		 LMC_OWNER_IDENTITY_VERSION) &
		((OwnershipPreemptedIdentityState[
		  LMC_OWNER_PREEMPT_HEADER_BASE + 1]$UDINT and 0xFFFE0000) = 0);
	if (expectedAdmissionMode = LMC_OWNER_ADMISSION_SAFETY) &
	   (OwnershipPreemptedIdentityState[
	    LMC_OWNER_PREEMPT_HEADER_BASE]$UDINT =
	    LMC_OWNER_PREEMPT_IDENTITY_MAGIC) &
	   (preemptRootValid = FALSE) then
		OwnershipState[24] := 1;
		Result := -3;
		RETURN;
	end_if;
	if (expectedAdmissionMode = LMC_OWNER_ADMISSION_SAFETY) &
	   (preemptRootValid = FALSE) then
		preemptBankValid := TRUE;
		identityIndex := 0;
		while identityIndex <= 323 do
			if OwnershipPreemptedState[identityIndex] <> 0 then
				preemptBankValid := FALSE;
			end_if;
			identityIndex += 1;
		end_while;
		identityIndex := 0;
		while identityIndex <= 431 do
			if OwnershipPreemptedIdentityState[identityIndex] <> 0 then
				preemptBankValid := FALSE;
			end_if;
			identityIndex += 1;
		end_while;
		if preemptBankValid = FALSE then
			OwnershipState[24] := 1;
			Result := -3;
			RETURN;
		end_if;
	end_if;
	preemptFlags := 0;
	cleanupRequiredMask := 0;
	cleanupCompleteMask := 0;
	if preemptRootValid then
		preemptFlags := OwnershipPreemptedIdentityState[
			LMC_OWNER_PREEMPT_HEADER_BASE + 1]$UDINT;
		cleanupRequiredMask := OwnershipPreemptedIdentityState[
			LMC_OWNER_PREEMPT_HEADER_BASE + 8]$UDINT;
		cleanupCompleteMask := OwnershipPreemptedIdentityState[
			LMC_OWNER_PREEMPT_HEADER_BASE + 9]$UDINT;
		if ((cleanupRequiredMask and (not AxisMask)) <> 0) |
		   ((cleanupCompleteMask and (not cleanupRequiredMask)) <> 0) then
			OwnershipState[24] := 1;
			Result := -3;
			RETURN;
		end_if;
		preemptBankValid := TRUE;
		preemptLmcFound := FALSE;
		preemptDs402Found := FALSE;
		preemptEncoderFound := FALSE;
		axisIndex := 1;
		while axisIndex <= LMC_OWNER_AXIS_COUNT do
			case axisIndex of
				1: axisBit := 0x00000001;
				2: axisBit := 0x00000002;
				3: axisBit := 0x00000004;
				4: axisBit := 0x00000008;
				5: axisBit := 0x00000010;
				6: axisBit := 0x00000020;
				7: axisBit := 0x00000040;
				8: axisBit := 0x00000080;
				9: axisBit := 0x00000100;
			else
				axisBit := 0;
			end_case;
			preemptRecordBase := (axisIndex - 1) * LMC_OWNER_AXIS_STRIDE;
			if (OwnershipPreemptedState[preemptRecordBase] <> axisIndex) |
			   (OwnershipPreemptedState[preemptRecordBase + 35]$UDINT <>
			    (LMC_OWNER_AXIS_RECORD_MAGIC + TO_UDINT(axisIndex))) then
				preemptBankValid := FALSE;
			end_if;
			if (AxisMask and axisBit) <> 0 then
				preemptState := OwnershipPreemptedState[preemptRecordBase + 1];
				preemptOwnerKind :=
					OwnershipPreemptedState[preemptRecordBase + 2];
				preemptCommand := OwnershipPreemptedState[preemptRecordBase + 3];
				preemptToken :=
					OwnershipPreemptedState[preemptRecordBase + 4]$UDINT;
				preemptGeneration :=
					OwnershipPreemptedState[preemptRecordBase + 5]$UDINT;
				preemptSession :=
					OwnershipPreemptedState[preemptRecordBase + 6]$UDINT;
				preemptSequence :=
					OwnershipPreemptedState[preemptRecordBase + 7]$UDINT;
				preemptMask :=
					OwnershipPreemptedState[preemptRecordBase + 11]$UDINT;
				preemptReference :=
					OwnershipPreemptedState[preemptRecordBase + 12];
				preemptResourceKind :=
					OwnershipPreemptedState[preemptRecordBase + 13];
				preemptAdmission :=
					OwnershipPreemptedState[preemptRecordBase + 14];
				preemptIdentitySize :=
					OwnershipPreemptedState[preemptRecordBase + 15]$UDINT;
				preemptSpecialValid := FALSE;
				case preemptOwnerKind of
					LMC_OWNER_KIND_LMC_HOME:
						preemptSpecialValid :=
							(preemptCommand = 0x7D13) &
							(preemptResourceKind =
							 LMC_OWNER_RESOURCE_LMC_HOME_ENGINE) &
							(preemptAdmission =
							 LMC_OWNER_ADMISSION_LIFECYCLE) &
							((preemptState = LMC_OWNER_STATE_RESERVED) |
							 (preemptState =
							  LMC_OWNER_STATE_LMC_HOME_ACTIVE)) &
							(preemptIdentitySize = 56);
					LMC_OWNER_KIND_DS402_HOME:
						preemptSpecialValid :=
							(preemptCommand = 0x7D15) &
							(preemptResourceKind =
							 LMC_OWNER_RESOURCE_DS402_HOME_ENGINE) &
							(preemptAdmission =
							 LMC_OWNER_ADMISSION_LIFECYCLE) &
							((preemptState = LMC_OWNER_STATE_RESERVED) |
							 (preemptState =
							  LMC_OWNER_STATE_DS402_HOME_ACTIVE)) &
							(preemptIdentitySize = 72);
					LMC_OWNER_KIND_ENCODER:
						preemptSpecialValid :=
							(preemptCommand = 0x7E53) &
							(preemptResourceKind =
							 LMC_OWNER_RESOURCE_DIAGNOSTICS_SDO_ENGINE) &
							(preemptAdmission =
							 LMC_OWNER_ADMISSION_LIFECYCLE) &
							((preemptState = LMC_OWNER_STATE_RESERVED) |
							 (preemptState = LMC_OWNER_STATE_TW20_QUEUED) |
							 (preemptState = LMC_OWNER_STATE_TW20_RUNNING) |
							 (preemptState = LMC_OWNER_STATE_TW20_DRAINING)) &
							(preemptIdentitySize = 72);
				else
				end_case;
				if preemptSpecialValid then
					case preemptResourceKind of
						LMC_OWNER_RESOURCE_LMC_HOME_ENGINE:
							if preemptLmcFound then
								preemptBankValid := FALSE;
							end_if;
							preemptLmcFound := TRUE;
						LMC_OWNER_RESOURCE_DS402_HOME_ENGINE:
							if preemptDs402Found then
								preemptBankValid := FALSE;
							end_if;
							preemptDs402Found := TRUE;
						LMC_OWNER_RESOURCE_DIAGNOSTICS_SDO_ENGINE:
							if preemptEncoderFound then
								preemptBankValid := FALSE;
							end_if;
							preemptEncoderFound := TRUE;
					else
						preemptBankValid := FALSE;
					end_case;
					if (preemptToken = 0) | (preemptGeneration = 0) |
					   (preemptSession = 0) | (preemptSequence = 0) |
					   (preemptMask <> axisBit) |
					   (preemptReference <> axisIndex) |
					   ((cleanupRequiredMask and axisBit) = 0) then
						preemptBankValid := FALSE;
					end_if;
					if (cleanupCompleteMask and axisBit) = 0 then
						case preemptResourceKind of
							LMC_OWNER_RESOURCE_LMC_HOME_ENGINE:
								preemptBankValid := preemptBankValid &
									(OwnershipState[7]$UDINT = preemptToken) &
									(OwnershipState[8]$UDINT =
									 preemptGeneration) &
									(OwnershipState[9]$UDINT = axisBit);
							LMC_OWNER_RESOURCE_DS402_HOME_ENGINE:
								preemptBankValid := preemptBankValid &
									(OwnershipState[10]$UDINT = preemptToken) &
									(OwnershipState[11]$UDINT =
									 preemptGeneration) &
									(OwnershipState[12]$UDINT = axisBit);
							LMC_OWNER_RESOURCE_DIAGNOSTICS_SDO_ENGINE:
								preemptBankValid := preemptBankValid &
									(OwnershipState[13]$UDINT = preemptToken) &
									(OwnershipState[14]$UDINT =
									 preemptGeneration) &
									(OwnershipState[15]$UDINT = axisBit);
						else
							preemptBankValid := FALSE;
						end_case;
					else
						singletonToken := 0;
						singletonGeneration := 0;
						singletonMask := 0;
						case preemptResourceKind of
							LMC_OWNER_RESOURCE_LMC_HOME_ENGINE:
								singletonToken := OwnershipState[7]$UDINT;
								singletonGeneration := OwnershipState[8]$UDINT;
								singletonMask := OwnershipState[9]$UDINT;
							LMC_OWNER_RESOURCE_DS402_HOME_ENGINE:
								singletonToken := OwnershipState[10]$UDINT;
								singletonGeneration := OwnershipState[11]$UDINT;
								singletonMask := OwnershipState[12]$UDINT;
							LMC_OWNER_RESOURCE_DIAGNOSTICS_SDO_ENGINE:
								singletonToken := OwnershipState[13]$UDINT;
								singletonGeneration := OwnershipState[14]$UDINT;
								singletonMask := OwnershipState[15]$UDINT;
						else
							preemptBankValid := FALSE;
						end_case;
						replacementValid := (singletonToken = 0) &
							(singletonGeneration = 0) & (singletonMask = 0);
						if replacementValid = FALSE then
							replacementValid :=
								(singletonToken <> 0) &
								(singletonGeneration <> 0) &
								(singletonMask <> 0) &
								(singletonMask <= LMC_OWNER_PROFILE_AXIS_MASK) &
								((singletonMask and (singletonMask - 1)) = 0) &
								(singletonToken <> preemptToken) &
								(singletonGeneration <> preemptGeneration);
							replacementFound := FALSE;
							probeAxisIndex := 1;
							while probeAxisIndex <= LMC_OWNER_AXIS_COUNT do
								case probeAxisIndex of
									1: probeAxisBit := 0x00000001;
									2: probeAxisBit := 0x00000002;
									3: probeAxisBit := 0x00000004;
									4: probeAxisBit := 0x00000008;
									5: probeAxisBit := 0x00000010;
									6: probeAxisBit := 0x00000020;
									7: probeAxisBit := 0x00000040;
									8: probeAxisBit := 0x00000080;
									9: probeAxisBit := 0x00000100;
								else
									probeAxisBit := 0;
								end_case;
								replacementRecordBase := LMC_OWNER_GLOBAL_SLOTS +
									((probeAxisIndex - 1) * LMC_OWNER_AXIS_STRIDE);
								if singletonMask = probeAxisBit then
									if replacementFound then
										replacementValid := FALSE;
									end_if;
									replacementFound := TRUE;
									replacementStateValid := FALSE;
									case preemptOwnerKind of
										LMC_OWNER_KIND_LMC_HOME:
											replacementStateValid :=
												(OwnershipState[replacementRecordBase + 1] =
												 LMC_OWNER_STATE_RESERVED) |
												(OwnershipState[replacementRecordBase + 1] =
												 LMC_OWNER_STATE_LMC_HOME_ACTIVE) |
												(OwnershipState[replacementRecordBase + 1] =
												 LMC_OWNER_STATE_QUARANTINED);
										LMC_OWNER_KIND_DS402_HOME:
											replacementStateValid :=
												(OwnershipState[replacementRecordBase + 1] =
												 LMC_OWNER_STATE_RESERVED) |
												(OwnershipState[replacementRecordBase + 1] =
												 LMC_OWNER_STATE_DS402_HOME_ACTIVE) |
												(OwnershipState[replacementRecordBase + 1] =
												 LMC_OWNER_STATE_QUARANTINED);
										LMC_OWNER_KIND_ENCODER:
											replacementStateValid :=
												(OwnershipState[replacementRecordBase + 1] =
												 LMC_OWNER_STATE_RESERVED) |
												(OwnershipState[replacementRecordBase + 1] =
												 LMC_OWNER_STATE_TW20_QUEUED) |
												(OwnershipState[replacementRecordBase + 1] =
												 LMC_OWNER_STATE_TW20_RUNNING) |
												(OwnershipState[replacementRecordBase + 1] =
												 LMC_OWNER_STATE_TW20_DRAINING) |
												(OwnershipState[replacementRecordBase + 1] =
												 LMC_OWNER_STATE_QUARANTINED);
									else
									end_case;
									replacementIdentitySize := preemptIdentitySize;
									replacementTailSize := 0;
									if replacementIdentitySize >
									   LMC_OWNER_IDENTITY_PREFIX_BYTES then
										replacementTailSize := replacementIdentitySize -
											LMC_OWNER_IDENTITY_PREFIX_BYTES;
									end_if;
									replacementTailOffset :=
										TO_UDINT(probeAxisIndex - 1) * 8;
									replacementPackedCommand :=
										TO_UDINT(preemptCommand) or
										(TO_UDINT(probeAxisIndex) shl 16);
									replacementPackedOwner :=
										TO_UDINT(preemptOwnerKind) or
										(TO_UDINT(preemptResourceKind) shl 8) or
										(TO_UDINT(LMC_OWNER_ADMISSION_LIFECYCLE) shl 16);
									replacementHeaderBase :=
										LMC_OWNER_IDENTITY_AXIS_HEADER_BASE +
										((probeAxisIndex - 1) *
										 LMC_OWNER_IDENTITY_AXIS_HEADER_STRIDE);
									replacementValid := replacementValid &
										replacementStateValid &
										(OwnershipState[replacementRecordBase] =
										 probeAxisIndex) &
										(OwnershipState[replacementRecordBase + 35]$UDINT =
										 (LMC_OWNER_AXIS_RECORD_MAGIC +
										  TO_UDINT(probeAxisIndex))) &
										(OwnershipState[replacementRecordBase + 2] =
										 preemptOwnerKind) &
										(OwnershipState[replacementRecordBase + 3] =
										 preemptCommand) &
										(OwnershipState[replacementRecordBase + 4]$UDINT =
										 singletonToken) &
										(OwnershipState[replacementRecordBase + 5]$UDINT =
										 singletonGeneration) &
										(OwnershipState[replacementRecordBase + 6]$UDINT <> 0) &
										(OwnershipState[replacementRecordBase + 7]$UDINT <> 0) &
										(OwnershipState[replacementRecordBase + 11]$UDINT =
										 singletonMask) &
										(OwnershipState[replacementRecordBase + 12] =
										 probeAxisIndex) &
										(OwnershipState[replacementRecordBase + 13] =
										 preemptResourceKind) &
										(OwnershipState[replacementRecordBase + 14] =
										 LMC_OWNER_ADMISSION_LIFECYCLE) &
										(OwnershipState[replacementRecordBase + 15]$UDINT =
										 replacementIdentitySize) &
										(OwnershipIdentityState[replacementHeaderBase]$UDINT =
										 (LMC_OWNER_IDENTITY_AXIS_MAGIC +
										  TO_UDINT(probeAxisIndex))) &
										(OwnershipIdentityState[replacementHeaderBase + 1] =
										 LMC_OWNER_IDENTITY_VERSION) &
										(OwnershipIdentityState[replacementHeaderBase + 2]$UDINT =
										 replacementIdentitySize) &
										(OwnershipIdentityState[replacementHeaderBase + 3]$UDINT =
										 singletonToken) &
										(OwnershipIdentityState[replacementHeaderBase + 4]$UDINT =
										 singletonGeneration) &
										(OwnershipIdentityState[replacementHeaderBase + 5]$UDINT =
										 singletonMask) &
										(OwnershipIdentityState[replacementHeaderBase + 6]$UDINT =
										 OwnershipState[replacementRecordBase + 6]$UDINT) &
										(OwnershipIdentityState[replacementHeaderBase + 7]$UDINT =
										 OwnershipState[replacementRecordBase + 7]$UDINT) &
										(OwnershipIdentityState[replacementHeaderBase + 8]$UDINT =
										 replacementPackedCommand) &
										(OwnershipIdentityState[replacementHeaderBase + 9]$UDINT =
										 replacementPackedOwner) &
										(OwnershipIdentityState[replacementHeaderBase + 10]$UDINT =
										 replacementTailOffset) &
										(OwnershipIdentityState[replacementHeaderBase + 11]$UDINT =
										 replacementTailSize);
									if replacementIdentitySize = 56 then
										replacementValid := replacementValid &
											(OwnershipState[replacementRecordBase + 30] = 0) &
											(OwnershipState[replacementRecordBase + 31] = 0);
									end_if;
								elsif (OwnershipState[replacementRecordBase + 4]$UDINT =
								       singletonToken) |
								      (OwnershipState[replacementRecordBase + 5]$UDINT =
								       singletonGeneration) then
									replacementValid := FALSE;
								end_if;
								probeAxisIndex += 1;
							end_while;
							replacementValid := replacementValid & replacementFound;
						end_if;
						probeAxisIndex := 1;
						while probeAxisIndex <= LMC_OWNER_AXIS_COUNT do
							replacementRecordBase := LMC_OWNER_GLOBAL_SLOTS +
								((probeAxisIndex - 1) * LMC_OWNER_AXIS_STRIDE);
							if (OwnershipState[replacementRecordBase + 4]$UDINT =
							    preemptToken) |
							   (OwnershipState[replacementRecordBase + 5]$UDINT =
							    preemptGeneration) then
								replacementValid := FALSE;
							end_if;
							probeAxisIndex += 1;
						end_while;
						if replacementValid = FALSE then
							preemptBankValid := FALSE;
						end_if;
					end_if;
					probeAxisIndex := 1;
					while probeAxisIndex <= LMC_OWNER_AXIS_COUNT do
						probeRecordBase := (probeAxisIndex - 1) *
							LMC_OWNER_AXIS_STRIDE;
						if (probeAxisIndex <> axisIndex) &
						   ((OwnershipPreemptedState[
						     probeRecordBase + 4]$UDINT = preemptToken) |
						    (OwnershipPreemptedState[
						     probeRecordBase + 5]$UDINT =
						     preemptGeneration)) then
							preemptBankValid := FALSE;
						end_if;
						probeAxisIndex += 1;
					end_while;
				elsif (cleanupRequiredMask and axisBit) <> 0 then
					preemptBankValid := FALSE;
				end_if;
			end_if;
			axisIndex += 1;
		end_while;
		if preemptBankValid = FALSE then
			OwnershipState[24] := 1;
			Result := -3;
			RETURN;
		end_if;
	end_if;
	cleanupReady := (cleanupCompleteMask and cleanupRequiredMask) =
		cleanupRequiredMask;
	forceQuarantine :=
		(preemptFlags and LMC_OWNER_PREEMPT_FLAG_FORCE_QUARANTINE) <> 0;
	axisIndex := 1;
	while axisIndex <= LMC_OWNER_AXIS_COUNT do
		case axisIndex of
			1: axisBit := 0x00000001;
			2: axisBit := 0x00000002;
			3: axisBit := 0x00000004;
			4: axisBit := 0x00000008;
			5: axisBit := 0x00000010;
			6: axisBit := 0x00000020;
			7: axisBit := 0x00000040;
			8: axisBit := 0x00000080;
			9: axisBit := 0x00000100;
		else
			axisBit := 0;
		end_case;
		if (AxisMask and axisBit) <> 0 then
			observerBase := (axisIndex - 1) * LMC_OWNER_OBSERVER_STRIDE;
			if (OwnershipObserverState[observerBase + 5]$UDINT and
			    LMC_OWNER_OBSERVER_FORCE_QUARANTINE) <> 0 then
				forceQuarantine := TRUE;
			end_if;
		end_if;
		axisIndex += 1;
	end_while;
	if (ReportKind = LMC_OWNER_REPORT_TERMINAL_SUCCESS) &
	   (expectedAdmissionMode = LMC_OWNER_ADMISSION_SAFETY) &
	   (cleanupReady = FALSE) then
		forceQuarantine := TRUE;
	end_if;
	restoreLease :=
		(ReportKind = LMC_OWNER_REPORT_TERMINAL_SUCCESS) &
		(forceQuarantine = FALSE) &
		(expectedOwnerKind = LMC_OWNER_KIND_GROUP) &
		((expectedCommandId = 0x20A4) |
		 (expectedCommandId = 0x7D22) |
		 (expectedCommandId = 0x2085));
	if restoreLease then
		// The lease header is preserved in its bank. Prove the complete exact
		// 0x2047 lease, selected records, one-byte identity, and zero suffix
		// before the first live ownership mutation.
		leaseValid :=
			(AxisMask = LMC_OWNER_PROFILE_AXIS_MASK) &
			(OwnershipLeaseIdentityState[
			 LMC_OWNER_LEASE_IDENTITY_HEADER_BASE]$UDINT =
			 LMC_OWNER_LEASE_IDENTITY_MAGIC) &
			(OwnershipLeaseIdentityState[
			 LMC_OWNER_LEASE_IDENTITY_HEADER_BASE + 1] =
			 LMC_OWNER_IDENTITY_VERSION) &
			(OwnershipLeaseIdentityState[
			 LMC_OWNER_LEASE_IDENTITY_HEADER_BASE + 2]$UDINT = 1) &
			(OwnershipLeaseIdentityState[
			 LMC_OWNER_LEASE_IDENTITY_HEADER_BASE + 3]$UDINT <> 0) &
			(OwnershipLeaseIdentityState[
			 LMC_OWNER_LEASE_IDENTITY_HEADER_BASE + 4]$UDINT <> 0) &
			(OwnershipLeaseIdentityState[
			 LMC_OWNER_LEASE_IDENTITY_HEADER_BASE + 5]$UDINT = AxisMask) &
			(OwnershipLeaseIdentityState[
			 LMC_OWNER_LEASE_IDENTITY_HEADER_BASE + 6]$UDINT <> 0) &
			(OwnershipLeaseIdentityState[
			 LMC_OWNER_LEASE_IDENTITY_HEADER_BASE + 7]$UDINT <> 0) &
			(OwnershipLeaseIdentityState[
			 LMC_OWNER_LEASE_IDENTITY_HEADER_BASE + 8]$UDINT =
			 (TO_UDINT(0x2047) or (TO_UDINT(0x0100) shl 16))) &
			(OwnershipLeaseIdentityState[
			 LMC_OWNER_LEASE_IDENTITY_HEADER_BASE + 9]$UDINT =
			 (TO_UDINT(LMC_OWNER_KIND_GROUP) or
			  (TO_UDINT(LMC_OWNER_RESOURCE_AXIS) shl 8) or
			  (TO_UDINT(LMC_OWNER_ADMISSION_ORDINARY) shl 16)));
		leaseFirstRecordBase := -1;
		axisIndex := 1;
		while axisIndex <= LMC_OWNER_AXIS_COUNT do
			case axisIndex of
				1: axisBit := 0x00000001;
				2: axisBit := 0x00000002;
				3: axisBit := 0x00000004;
				4: axisBit := 0x00000008;
				5: axisBit := 0x00000010;
				6: axisBit := 0x00000020;
				7: axisBit := 0x00000040;
				8: axisBit := 0x00000080;
				9: axisBit := 0x00000100;
			else
				axisBit := 0;
			end_case;
			leaseRecordBase := (axisIndex - 1) * LMC_OWNER_AXIS_STRIDE;
			if (OwnershipLeaseState[leaseRecordBase] <> axisIndex) |
			   (OwnershipLeaseState[leaseRecordBase + 35]$UDINT <>
			    (LMC_OWNER_AXIS_RECORD_MAGIC + TO_UDINT(axisIndex))) then
				leaseValid := FALSE;
			end_if;
			if (AxisMask and axisBit) <> 0 then
				if (OwnershipLeaseState[leaseRecordBase + 1] <>
				    LMC_OWNER_STATE_GROUP_LEASE) |
				   (OwnershipLeaseState[leaseRecordBase + 2] <>
				    LMC_OWNER_KIND_GROUP) |
				   (OwnershipLeaseState[leaseRecordBase + 3] <> 0x2047) |
				   (OwnershipLeaseState[leaseRecordBase + 4]$UDINT <>
				    OwnershipLeaseIdentityState[
				     LMC_OWNER_LEASE_IDENTITY_HEADER_BASE + 3]$UDINT) |
				   (OwnershipLeaseState[leaseRecordBase + 5]$UDINT <>
				    OwnershipLeaseIdentityState[
				     LMC_OWNER_LEASE_IDENTITY_HEADER_BASE + 4]$UDINT) |
				   (OwnershipLeaseState[leaseRecordBase + 6]$UDINT <>
				    OwnershipLeaseIdentityState[
				     LMC_OWNER_LEASE_IDENTITY_HEADER_BASE + 6]$UDINT) |
				   (OwnershipLeaseState[leaseRecordBase + 7]$UDINT <>
				    OwnershipLeaseIdentityState[
				     LMC_OWNER_LEASE_IDENTITY_HEADER_BASE + 7]$UDINT) |
				   (OwnershipLeaseState[leaseRecordBase + 11]$UDINT <> AxisMask) |
				   (OwnershipLeaseState[leaseRecordBase + 12] <> 0x0100) |
				   (OwnershipLeaseState[leaseRecordBase + 13] <>
				    LMC_OWNER_RESOURCE_AXIS) |
				   (OwnershipLeaseState[leaseRecordBase + 14] <>
				    LMC_OWNER_ADMISSION_ORDINARY) |
				   (OwnershipLeaseState[leaseRecordBase + 15]$UDINT <> 1) |
				   (OwnershipLeaseState[leaseRecordBase + 16]$UDINT <> 1) then
					leaseValid := FALSE;
				end_if;
				identityIndex := 17;
				while identityIndex <= 31 do
					if OwnershipLeaseState[leaseRecordBase + identityIndex] <> 0 then
						leaseValid := FALSE;
					end_if;
					identityIndex += 1;
				end_while;
				if leaseFirstRecordBase < 0 then
					leaseFirstRecordBase := leaseRecordBase;
				else
					identityCompareResult := _memcmp(
						ptr1:=#OwnershipLeaseState[leaseFirstRecordBase + 16],
						ptr2:=#OwnershipLeaseState[leaseRecordBase + 16], cntr:=1);
					if identityCompareResult <> 0 then
						leaseValid := FALSE;
					end_if;
				end_if;
			else
				if (OwnershipLeaseState[leaseRecordBase + 4]$UDINT =
				    OwnershipLeaseIdentityState[
				     LMC_OWNER_LEASE_IDENTITY_HEADER_BASE + 3]$UDINT) |
				   (OwnershipLeaseState[leaseRecordBase + 5]$UDINT =
				    OwnershipLeaseIdentityState[
				     LMC_OWNER_LEASE_IDENTITY_HEADER_BASE + 4]$UDINT) then
					leaseValid := FALSE;
				end_if;
				identityIndex := 1;
				while identityIndex <= 34 do
					if OwnershipLeaseState[leaseRecordBase + identityIndex] <> 0 then
						leaseValid := FALSE;
					end_if;
					identityIndex += 1;
				end_while;
			end_if;
			axisIndex += 1;
		end_while;
		identityIndex := 0;
		while identityIndex < LMC_OWNER_IDENTITY_SUFFIX_DINTS do
			if OwnershipLeaseIdentityState[identityIndex] <> 0 then
				leaseValid := FALSE;
			end_if;
			identityIndex += 1;
		end_while;
		if leaseValid = FALSE then
			OwnershipState[24] := 1;
			Result := -3;
			RETURN;
		end_if;
	end_if;
	destroyBanks :=
		(ReportKind = LMC_OWNER_REPORT_TERMINAL_SUCCESS) &
		((expectedCommandId = 0x2048) | (expectedCommandId = 0x204B));
	retainGroupLease :=
		(ReportKind = LMC_OWNER_REPORT_TERMINAL_SUCCESS) &
		(forceQuarantine = FALSE) &
		(expectedOwnerKind = LMC_OWNER_KIND_GROUP) &
		(expectedCommandId = 0x2047);
	if retainGroupLease then
		// A successful GroupEnable establishes its own accepted exact lease;
		// it does not restore or synthesize a prior lease record.
		retainLeaseValid :=
			(expectedResourceKind = LMC_OWNER_RESOURCE_AXIS) &
			(expectedAdmissionMode = LMC_OWNER_ADMISSION_ORDINARY) &
			(expectedReference = 0x0100) &
			(AxisMask = LMC_OWNER_PROFILE_AXIS_MASK) &
			(expectedSession <> 0) & (expectedSequence <> 0) &
			(identitySize = 1) &
			(OwnershipIdentityState[
			 LMC_OWNER_IDENTITY_GROUP_HEADER_BASE]$UDINT =
			 LMC_OWNER_IDENTITY_GROUP_MAGIC) &
			(OwnershipIdentityState[
			 LMC_OWNER_IDENTITY_GROUP_HEADER_BASE + 1] =
			 LMC_OWNER_IDENTITY_VERSION) &
			(OwnershipIdentityState[
			 LMC_OWNER_IDENTITY_GROUP_HEADER_BASE + 2]$UDINT = 1) &
			(OwnershipIdentityState[
			 LMC_OWNER_IDENTITY_GROUP_HEADER_BASE + 3]$UDINT =
			 AdmissionToken) &
			(OwnershipIdentityState[
			 LMC_OWNER_IDENTITY_GROUP_HEADER_BASE + 4]$UDINT =
			 OwnerGeneration) &
			(OwnershipIdentityState[
			 LMC_OWNER_IDENTITY_GROUP_HEADER_BASE + 5]$UDINT = AxisMask) &
			(OwnershipIdentityState[
			 LMC_OWNER_IDENTITY_GROUP_HEADER_BASE + 6]$UDINT =
			 expectedSession) &
			(OwnershipIdentityState[
			 LMC_OWNER_IDENTITY_GROUP_HEADER_BASE + 7]$UDINT =
			 expectedSequence) &
			(OwnershipIdentityState[
			 LMC_OWNER_IDENTITY_GROUP_HEADER_BASE + 8]$UDINT =
			 (TO_UDINT(0x2047) or (TO_UDINT(0x0100) shl 16))) &
			(OwnershipIdentityState[
			 LMC_OWNER_IDENTITY_GROUP_HEADER_BASE + 9]$UDINT =
			 (TO_UDINT(LMC_OWNER_KIND_GROUP) or
			  (TO_UDINT(LMC_OWNER_RESOURCE_AXIS) shl 8) or
			  (TO_UDINT(LMC_OWNER_ADMISSION_ORDINARY) shl 16)));
		axisIndex := 1;
		while axisIndex <= LMC_OWNER_AXIS_COUNT do
			case axisIndex of
				1: axisBit := 0x00000001;
				2: axisBit := 0x00000002;
				3: axisBit := 0x00000004;
				4: axisBit := 0x00000008;
				5: axisBit := 0x00000010;
				6: axisBit := 0x00000020;
				7: axisBit := 0x00000040;
				8: axisBit := 0x00000080;
				9: axisBit := 0x00000100;
			else
				axisBit := 0;
			end_case;
			if (AxisMask and axisBit) <> 0 then
				recordBase := LMC_OWNER_GLOBAL_SLOTS +
					((axisIndex - 1) * LMC_OWNER_AXIS_STRIDE);
				if OwnershipState[recordBase + 16]$UDINT <> 1 then
					retainLeaseValid := FALSE;
				end_if;
				identityIndex := 17;
				while identityIndex <= 31 do
					if OwnershipState[recordBase + identityIndex] <> 0 then
						retainLeaseValid := FALSE;
					end_if;
					identityIndex += 1;
				end_while;
				identityCompareResult := _memcmp(
					ptr1:=#OwnershipState[firstRecordBase + 16],
					ptr2:=#OwnershipState[recordBase + 16], cntr:=1);
				if identityCompareResult <> 0 then
					retainLeaseValid := FALSE;
				end_if;
			end_if;
			axisIndex += 1;
		end_while;
		identityIndex := 0;
		while identityIndex < LMC_OWNER_IDENTITY_SUFFIX_DINTS do
			if OwnershipIdentityState[identityIndex] <> 0 then
				retainLeaseValid := FALSE;
			end_if;
			identityIndex += 1;
		end_while;
		if retainLeaseValid = FALSE then
			OwnershipState[24] := 1;
			Result := -3;
			RETURN;
		end_if;
	end_if;
	clearOwner :=
		(ReportKind = LMC_OWNER_REPORT_TERMINAL_SUCCESS) &
		(forceQuarantine = FALSE) &
		(restoreLease = FALSE) & (retainGroupLease = FALSE);
	if ReportKind = LMC_OWNER_REPORT_TERMINAL_SAFE_FAILURE then
		clearOwner := (expectedOwnerKind <> LMC_OWNER_KIND_DIRECT) &
			(expectedOwnerKind <> LMC_OWNER_KIND_GROUP) &
			(forceQuarantine = FALSE);
	end_if;
	if (expectedCommandId = 0x7D13) &
	   (expectedOwnerKind = LMC_OWNER_KIND_LMC_HOME) &
	   (expectedResourceKind = LMC_OWNER_RESOURCE_LMC_HOME_ENGINE) &
	   (expectedAdmissionMode = LMC_OWNER_ADMISSION_LIFECYCLE) &
	   (preemptRootValid = FALSE) & (forceQuarantine = FALSE) &
	   clearOwner &
	   ((ReportKind = LMC_OWNER_REPORT_TERMINAL_SUCCESS) |
	    (ReportKind = LMC_OWNER_REPORT_TERMINAL_SAFE_FAILURE)) then
		// Publish an immutable exact receipt before any owner surface is cleared.
		// The caller accepts the receipt and replays this call to perform cleanup.
		homeReceiptAxisMaskValid := FALSE;
		case expectedReference of
			1: homeReceiptAxisMaskValid := AxisMask = 0x00000001;
			2: homeReceiptAxisMaskValid := AxisMask = 0x00000002;
			3: homeReceiptAxisMaskValid := AxisMask = 0x00000004;
			4: homeReceiptAxisMaskValid := AxisMask = 0x00000008;
		else
		end_case;
		if (homeReceiptAxisMaskValid = FALSE) |
		   (ZeroHomeState[51]$UDINT <> LMC_HOME_RECORD_MAGIC) |
		   (ZeroHomeState[33]$UDINT = 0) |
		   (ZeroHomeState[34]$UDINT <> AdmissionToken) |
		   (ZeroHomeState[35]$UDINT <> OwnerGeneration) |
		   (ZeroHomeState[36]$UDINT <> expectedSession) |
		   (ZeroHomeState[37]$UDINT <> expectedSequence) |
		   (ZeroHomeState[38]$UDINT <> AxisMask) |
		   (ZeroHomeState[39] <> LMC_HOME_ENGINE_FINALIZE) |
		   (ZeroHomeState[57]$UDINT <> ReportValue0) |
		   (ZeroHomeState[58] <> TO_DINT(ReportKind)) |
		   (ZeroHomeState[59] <> 0) |
		   (ZeroHomeState[31]$UDINT <> ReportValue1) |
		   (ZeroHomeState[46]$UDINT <> ObservationCycle) |
		   ((ZeroHomeState[56]$UDINT and
		     LMC_HOME_FLAG_OWNER_FINALIZE_INTENT) = 0) |
		   ((ZeroHomeState[56]$UDINT and
		     LMC_HOME_FLAG_OWNER_FINALIZE_ACCEPTED) <> 0) |
		   (ZeroHomeState[60] <> 0) then
			OwnershipState[24] := 1;
			Result := -3;
			RETURN;
		end_if;
		ZeroHomeState[60] := 0;
		ZeroHomeState[61] := LMC_HOME_OWNER_RECEIPT_PREPARED;
		ZeroHomeState[62] := 0;
		ZeroHomeState[63]$UDINT := ZeroHomeState[33]$UDINT;
		ZeroHomeState[60]$UDINT := LMC_HOME_OWNER_RECEIPT_MAGIC;
		Result := 0;
		RETURN;
	end_if;
	axisIndex := 1;
	while axisIndex <= LMC_OWNER_AXIS_COUNT do
		case axisIndex of
			1: axisBit := 0x00000001;
			2: axisBit := 0x00000002;
			3: axisBit := 0x00000004;
			4: axisBit := 0x00000008;
			5: axisBit := 0x00000010;
			6: axisBit := 0x00000020;
			7: axisBit := 0x00000040;
			8: axisBit := 0x00000080;
			9: axisBit := 0x00000100;
		else
			axisBit := 0;
		end_case;
		if (AxisMask and axisBit) <> 0 then
			recordBase := LMC_OWNER_GLOBAL_SLOTS +
				((axisIndex - 1) * LMC_OWNER_AXIS_STRIDE);
			observerBase := (axisIndex - 1) * LMC_OWNER_OBSERVER_STRIDE;
			OwnershipState[recordBase + 9]$UDINT := ObservationCycle;
			OwnershipState[recordBase + 32] := TO_DINT(ReportKind);
			OwnershipState[recordBase + 33]$UDINT := ReportValue0;
			OwnershipState[recordBase + 34]$UDINT := ReportValue1;
			case ReportKind of
				LMC_OWNER_REPORT_TERMINAL_SUCCESS:
					if forceQuarantine then
						OwnershipState[recordBase + 1] :=
							LMC_OWNER_STATE_QUARANTINED;
						OwnershipState[recordBase + 32] :=
							LMC_OWNER_REPORT_QUARANTINE;
					elsif restoreLease then
						// Exact lease restore is applied after this validation loop.
					elsif retainGroupLease then
						OwnershipState[recordBase + 1] :=
							LMC_OWNER_STATE_GROUP_LEASE;
						observerIndex := 0;
						while observerIndex < LMC_OWNER_OBSERVER_STRIDE do
							OwnershipObserverState[observerBase + observerIndex] := 0;
							observerIndex += 1;
						end_while;
					elsif clearOwner then
						_memset(dest:=#OwnershipState[recordBase], usByte:=0,
							cntr:=LMC_OWNER_AXIS_STRIDE * 4);
						OwnershipState[recordBase] := axisIndex;
						OwnershipState[recordBase + 35]$UDINT :=
							LMC_OWNER_AXIS_RECORD_MAGIC + TO_UDINT(axisIndex);
						_memset(dest:=#OwnershipObserverState[observerBase],
							usByte:=0, cntr:=LMC_OWNER_OBSERVER_STRIDE * 4);
					end_if;
				LMC_OWNER_REPORT_TERMINAL_SAFE_FAILURE:
					if (expectedOwnerKind = LMC_OWNER_KIND_DIRECT) |
					   (expectedOwnerKind = LMC_OWNER_KIND_GROUP) |
					   forceQuarantine then
						OwnershipState[recordBase + 1] :=
							LMC_OWNER_STATE_QUARANTINED;
					elsif clearOwner then
						_memset(dest:=#OwnershipState[recordBase], usByte:=0,
							cntr:=LMC_OWNER_AXIS_STRIDE * 4);
						OwnershipState[recordBase] := axisIndex;
						OwnershipState[recordBase + 35]$UDINT :=
							LMC_OWNER_AXIS_RECORD_MAGIC + TO_UDINT(axisIndex);
						_memset(dest:=#OwnershipObserverState[observerBase],
							usByte:=0, cntr:=LMC_OWNER_OBSERVER_STRIDE * 4);
					end_if;
				LMC_OWNER_REPORT_QUARANTINE:
					OwnershipState[recordBase + 1] :=
						LMC_OWNER_STATE_QUARANTINED;
				LMC_OWNER_REPORT_SAFETY_PREEMPT:
					OwnershipState[recordBase + 1] :=
						LMC_OWNER_STATE_SAFETY_PREEMPTING;
			else
			end_case;
		end_if;
		axisIndex += 1;
	end_while;

	if restoreLease then
		OwnershipIdentityState[
			LMC_OWNER_IDENTITY_GROUP_HEADER_BASE] := 0;
		_memcpy(ptr1:=#OwnershipIdentityState[0],
			ptr2:=#OwnershipLeaseIdentityState[0],
			cntr:=LMC_OWNER_IDENTITY_SUFFIX_BYTES);
		_memset(dest:=#OwnershipIdentityState[
			LMC_OWNER_IDENTITY_GROUP_HEADER_BASE], usByte:=0, cntr:=40);
		clearIndex := 1;
		while clearIndex <= 9 do
			OwnershipIdentityState[
				LMC_OWNER_IDENTITY_GROUP_HEADER_BASE + clearIndex] :=
				OwnershipLeaseIdentityState[
				 LMC_OWNER_LEASE_IDENTITY_HEADER_BASE + clearIndex];
			clearIndex += 1;
		end_while;
		axisIndex := 1;
		while axisIndex <= LMC_OWNER_AXIS_COUNT do
			case axisIndex of
				1: axisBit := 0x00000001;
				2: axisBit := 0x00000002;
				3: axisBit := 0x00000004;
				4: axisBit := 0x00000008;
				5: axisBit := 0x00000010;
				6: axisBit := 0x00000020;
				7: axisBit := 0x00000040;
				8: axisBit := 0x00000080;
				9: axisBit := 0x00000100;
			else
				axisBit := 0;
			end_case;
			if (AxisMask and axisBit) <> 0 then
				recordBase := LMC_OWNER_GLOBAL_SLOTS +
					((axisIndex - 1) * LMC_OWNER_AXIS_STRIDE);
				clearIndex := (axisIndex - 1) * LMC_OWNER_AXIS_STRIDE;
				observerBase := (axisIndex - 1) *
					LMC_OWNER_OBSERVER_STRIDE;
				identityTailOffset := LMC_OWNER_IDENTITY_AXIS_HEADER_BASE +
					TO_UDINT((axisIndex - 1) *
					 LMC_OWNER_IDENTITY_AXIS_HEADER_STRIDE);
				OwnershipIdentityState[TO_DINT(identityTailOffset)] := 0;
				_memset(dest:=#OwnershipIdentityState[
					TO_DINT(identityTailOffset)], usByte:=0,
					cntr:=LMC_OWNER_IDENTITY_AXIS_HEADER_STRIDE * 4);
				_memcpy(ptr1:=#OwnershipState[recordBase],
					ptr2:=#OwnershipLeaseState[clearIndex],
					cntr:=LMC_OWNER_AXIS_STRIDE * 4);
				_memset(dest:=#OwnershipObserverState[observerBase], usByte:=0,
					cntr:=LMC_OWNER_OBSERVER_STRIDE * 4);
			end_if;
			axisIndex += 1;
		end_while;
		OwnershipIdentityState[
			LMC_OWNER_IDENTITY_GROUP_HEADER_BASE]$UDINT :=
			LMC_OWNER_IDENTITY_GROUP_MAGIC;
	end_if;

	if clearOwner then
		axisIndex := 1;
		while axisIndex <= LMC_OWNER_AXIS_COUNT do
			case axisIndex of
				1: axisBit := 0x00000001;
				2: axisBit := 0x00000002;
				3: axisBit := 0x00000004;
				4: axisBit := 0x00000008;
				5: axisBit := 0x00000010;
				6: axisBit := 0x00000020;
				7: axisBit := 0x00000040;
				8: axisBit := 0x00000080;
				9: axisBit := 0x00000100;
			else
				axisBit := 0;
			end_case;
			if (AxisMask and axisBit) <> 0 then
				identityTailOffset := LMC_OWNER_IDENTITY_AXIS_HEADER_BASE +
					TO_UDINT((axisIndex - 1) *
					 LMC_OWNER_IDENTITY_AXIS_HEADER_STRIDE);
				_memset(dest:=#OwnershipIdentityState[
					TO_DINT(identityTailOffset)], usByte:=0,
					cntr:=LMC_OWNER_IDENTITY_AXIS_HEADER_STRIDE * 4);
			end_if;
			axisIndex += 1;
		end_while;
		if expectedOwnerKind = LMC_OWNER_KIND_GROUP then
			OwnershipIdentityState[
				LMC_OWNER_IDENTITY_GROUP_HEADER_BASE] := 0;
			if expectedAdmissionMode <> LMC_OWNER_ADMISSION_SAFETY then
				_memset(dest:=#OwnershipIdentityState[0], usByte:=0,
					cntr:=LMC_OWNER_IDENTITY_SUFFIX_BYTES);
			end_if;
			_memset(dest:=#OwnershipIdentityState[
				LMC_OWNER_IDENTITY_GROUP_HEADER_BASE], usByte:=0, cntr:=40);
		elsif identityTailSize > 0 then
			identityTailOffset := TO_UDINT(expectedReference - 1) * 8;
			_memset(dest:=#OwnershipIdentityState[
				TO_DINT(identityTailOffset / 4)], usByte:=0,
				cntr:=identityTailSize);
		end_if;
	end_if;

	if (ReportKind = LMC_OWNER_REPORT_TERMINAL_SUCCESS) &
	   (forceQuarantine = FALSE) then
		if preemptRootValid then
			OwnershipPreemptedIdentityState[
				LMC_OWNER_PREEMPT_HEADER_BASE] := 0;
			_memset(dest:=#OwnershipPreemptedState[0], usByte:=0,
				cntr:=sizeof(OwnershipPreemptedState));
			_memset(dest:=#OwnershipPreemptedIdentityState[0], usByte:=0,
				cntr:=sizeof(OwnershipPreemptedIdentityState));
		end_if;
		if restoreLease | destroyBanks then
			OwnershipLeaseIdentityState[
				LMC_OWNER_LEASE_IDENTITY_HEADER_BASE] := 0;
			_memset(dest:=#OwnershipLeaseState[0], usByte:=0,
				cntr:=sizeof(OwnershipLeaseState));
			_memset(dest:=#OwnershipLeaseIdentityState[0], usByte:=0,
				cntr:=sizeof(OwnershipLeaseIdentityState));
		end_if;
	end_if;

	if (ReportKind = LMC_OWNER_REPORT_TERMINAL_SUCCESS) |
	   (ReportKind = LMC_OWNER_REPORT_TERMINAL_SAFE_FAILURE) then
		if (OwnershipState[7]$UDINT = AdmissionToken) &
		   (OwnershipState[8]$UDINT = OwnerGeneration) then
			OwnershipState[7] := 0;
			OwnershipState[8] := 0;
			OwnershipState[9] := 0;
		end_if;
		if (OwnershipState[10]$UDINT = AdmissionToken) &
		   (OwnershipState[11]$UDINT = OwnerGeneration) then
			OwnershipState[10] := 0;
			OwnershipState[11] := 0;
			OwnershipState[12] := 0;
		end_if;
		if (OwnershipState[13]$UDINT = AdmissionToken) &
		   (OwnershipState[14]$UDINT = OwnerGeneration) then
			OwnershipState[13] := 0;
			OwnershipState[14] := 0;
			OwnershipState[15] := 0;
		end_if;
	end_if;
	Result := 0;

END_FUNCTION

FUNCTION GLOBAL LMCControlCommandService::ReconcileAxisOwnershipStartup
	VAR_INPUT
		DiagnosticsBootId 	: UDINT;
		ObservationCycle 	: UDINT;
		ReportCycle 	: UDINT;
		DiagnosticsDrainFlags 	: UDINT;
	END_VAR
	VAR_OUTPUT
		Result 	: DINT;
	END_VAR
	VAR
		startupSnapshot : ARRAY [0..11] OF UDINT;
		copyResult : DINT;
		axisIndex : DINT;
		recordBase : DINT;
		stateIndex : DINT;
		combinedProof : UDINT;
		groupSignature : UDINT;
		robotState : DINT;
		profileLockState : DINT;
		profileFinished : DINT;
		stableElapsedMilliseconds : UDINT;
		tableIdle : BOOL;
		physicalIdle : BOOL;
		groupIdle : BOOL;
		drained : BOOL;
		signatureStable : BOOL;
		freshObservation : BOOL;
		auxiliaryIdle : BOOL;
	END_VAR

	Result := -1;
	if (DiagnosticsBootId = 0) | (ObservationCycle = 0) |
		(ReportCycle = 0) then
		RETURN;
	end_if;

	// Normal operations may make a completed same-boot table non-idle. Do not
	// reinterpret those transient states as startup failures.
	if (OwnershipState[0]$UDINT = LMC_OWNER_TABLE_MAGIC) &
		(OwnershipState[3]$UDINT = DiagnosticsBootId) then
		if (OwnershipState[4]$UDINT <> 0) &
			(OwnershipState[5]$UDINT = LMC_OWNER_STARTUP_PROOF_REQUIRED) &
			(OwnershipState[6] = 0) &
			(OwnershipState[24] = 0) then
			Result := 0;
		else
			Result := -3;
		end_if;
		RETURN;
	end_if;

	auxiliaryIdle := TRUE;
	stateIndex := 0;
	while stateIndex <= 431 do
		if (OwnershipIdentityState[stateIndex] <> 0) |
		   (OwnershipPreemptedIdentityState[stateIndex] <> 0) then
			auxiliaryIdle := FALSE;
		end_if;
		stateIndex += 1;
	end_while;
	stateIndex := 0;
	while stateIndex <= 323 do
		if (OwnershipLeaseState[stateIndex] <> 0) |
		   (OwnershipPreemptedState[stateIndex] <> 0) |
		   (OwnershipLeaseIdentityState[stateIndex] <> 0) then
			auxiliaryIdle := FALSE;
		end_if;
		stateIndex += 1;
	end_while;
	if auxiliaryIdle = FALSE then
		Result := -3;
		RETURN;
	end_if;

	// A nonzero existing table may be replaced only when it is a valid,
	// prior-boot, completely idle owner table.
	if OwnershipState[0]$UDINT = 0 then
		tableIdle := TRUE;
		stateIndex := 1;
		while stateIndex <= 351 do
			if OwnershipState[stateIndex] <> 0 then
				tableIdle := FALSE;
			end_if;
			stateIndex += 1;
		end_while;
		if tableIdle = FALSE then
			Result := -3;
			RETURN;
		end_if;
	elsif OwnershipState[0]$UDINT = LMC_OWNER_TABLE_MAGIC then
		tableIdle := (OwnershipState[3]$UDINT <> 0) &
			(OwnershipState[4]$UDINT <> 0) &
			(OwnershipState[5]$UDINT = LMC_OWNER_STARTUP_PROOF_REQUIRED) &
			(OwnershipState[6] = 0) &
			(OwnershipState[7] = 0) & (OwnershipState[8] = 0) &
			(OwnershipState[9] = 0) & (OwnershipState[10] = 0) &
			(OwnershipState[11] = 0) & (OwnershipState[12] = 0) &
			(OwnershipState[13] = 0) & (OwnershipState[14] = 0) &
			(OwnershipState[15] = 0) & (OwnershipState[16] = 0) &
			(OwnershipState[17] = 0) & (OwnershipState[18] = 0) &
			(OwnershipState[19] = 0) & (OwnershipState[20] = 0) &
			(OwnershipState[21] = 0) & (OwnershipState[24] = 0) &
			(OwnershipState[25] = 0) & (OwnershipState[26] = 0) &
			(OwnershipState[27] = 0);
		axisIndex := 1;
		while axisIndex <= LMC_OWNER_AXIS_COUNT do
			recordBase := LMC_OWNER_GLOBAL_SLOTS +
				((axisIndex - 1) * LMC_OWNER_AXIS_STRIDE);
			if (OwnershipState[recordBase] <> axisIndex) |
				(OwnershipState[recordBase + 35]$UDINT <>
				 (LMC_OWNER_AXIS_RECORD_MAGIC + TO_UDINT(axisIndex))) then
				tableIdle := FALSE;
			end_if;
			stateIndex := 1;
			while stateIndex <= 34 do
				if OwnershipState[recordBase + stateIndex] <> 0 then
					tableIdle := FALSE;
				end_if;
				stateIndex += 1;
			end_while;
			axisIndex += 1;
		end_while;
		if tableIdle = FALSE then
			Result := -3;
			RETURN;
		end_if;
	else
		Result := -3;
		RETURN;
	end_if;

	if (OwnershipStartupState[0]$UDINT <> LMC_OWNER_STARTUP_STATE_MAGIC) |
		(OwnershipStartupState[1]$UDINT <> DiagnosticsBootId) then
		_memset(dest:=#OwnershipStartupState[0], usByte:=0, cntr:=64);
		OwnershipStartupState[0]$UDINT := LMC_OWNER_STARTUP_STATE_MAGIC;
		OwnershipStartupState[1]$UDINT := DiagnosticsBootId;
	end_if;

	Result := 1;
	if IsClientConnected(#InputLatch) = FALSE then
		OwnershipStartupState[3] := 0;
		OwnershipStartupState[4]$UDINT := 0x00000001;
		OwnershipStartupState[14] := 0;
		OwnershipStartupState[15] := 1;
		RETURN;
	end_if;
	copyResult := InputLatch.CopyAxisOwnershipStartupSnapshot(
		pDest:=#startupSnapshot[0], DestSize:=48);
	if copyResult <> 0 then
		OwnershipStartupState[3] := 0;
		OwnershipStartupState[4]$UDINT := 0x00000001;
		OwnershipStartupState[14] := 0;
		OwnershipStartupState[15] := 2;
		RETURN;
	end_if;
	if (startupSnapshot[0] <> LMC_OWNER_STARTUP_SNAPSHOT_MAGIC) |
		(startupSnapshot[1] = 0) |
		(startupSnapshot[1] <> ObservationCycle) |
		(startupSnapshot[11] <> 0) then
		OwnershipStartupState[3] := 0;
		OwnershipStartupState[14] := 0;
		OwnershipStartupState[15] := -1;
		Result := -1;
		RETURN;
	end_if;

	physicalIdle :=
		((startupSnapshot[10] and 0x00000001) <> 0) &
		((startupSnapshot[2] and LMC_AXIS_STATUS_STANDSTILL) <> 0) &
		((startupSnapshot[2] and LMC_OWNER_STARTUP_AXIS_CLEAR_MASK) = 0) &
		((startupSnapshot[3] and LMC_AXIS_STATUS_STANDSTILL) <> 0) &
		((startupSnapshot[3] and LMC_OWNER_STARTUP_AXIS_CLEAR_MASK) = 0) &
		((startupSnapshot[4] and LMC_AXIS_STATUS_STANDSTILL) <> 0) &
		((startupSnapshot[4] and LMC_OWNER_STARTUP_AXIS_CLEAR_MASK) = 0) &
		((startupSnapshot[5] and LMC_AXIS_STATUS_STANDSTILL) <> 0) &
		((startupSnapshot[5] and LMC_OWNER_STARTUP_AXIS_CLEAR_MASK) = 0);

	groupIdle := FALSE;
	groupSignature := 0;
	if (IsClientConnected(#LMCRobot) <> 0) &
		(IsClientConnected(#LMCAxis1) <> 0) &
		(IsClientConnected(#LMCAxis2) <> 0) &
		(IsClientConnected(#LMCAxis3) <> 0) &
		(IsClientConnected(#LMCAxis4) <> 0) then
		robotState := LMCRobot.ReadRobotParameter(ParNo:=_ROBOT_STATE, Mode:=0);
		profileLockState := LMCRobot.ReadProfileParameter(
			ParNo:=_LMCPROF_LockState);
		profileFinished := LMCRobot.ProfileInPosition(
			Mode:=_LMCPROF_ProfileFinished);
		groupSignature := (TO_UDINT(robotState) and 0x0000FFFF) or
			((TO_UDINT(profileLockState) and 0x000000FF) shl 16);
		if profileFinished <> 0 then
			groupSignature := groupSignature or 0x01000000;
		end_if;
		groupIdle := (profileLockState = 0) &
			((startupSnapshot[2] and LMC_OWNER_STARTUP_AXIS_LOCK_MASK) = 0) &
			((startupSnapshot[3] and LMC_OWNER_STARTUP_AXIS_LOCK_MASK) = 0) &
			((startupSnapshot[4] and LMC_OWNER_STARTUP_AXIS_LOCK_MASK) = 0) &
			((startupSnapshot[5] and LMC_OWNER_STARTUP_AXIS_LOCK_MASK) = 0) &
			((robotState = _ROBOT_PASSIVE$DINT) |
			 ((robotState = _ROBOT_DIRECT$DINT) & (profileFinished <> 0)));
	end_if;

	drained := (startupSnapshot[10] = LMC_OWNER_STARTUP_LATCH_REQUIRED) &
		(DiagnosticsDrainFlags = LMC_OWNER_STARTUP_DIAG_REQUIRED) &
		(ZeroHomeState[0] <> LMC_HOME_RECORD_RUNNING) &
		(ZeroHomeState[0] <> LMC_HOME_RECORD_QUARANTINED) &
		((ZeroHomeState[39] = LMC_HOME_ENGINE_IDLE) |
		 (ZeroHomeState[39] = LMC_HOME_ENGINE_TERMINAL));

	combinedProof := 0x00000001;
	if physicalIdle then
		combinedProof := combinedProof or 0x00000002;
	end_if;
	if groupIdle then
		combinedProof := combinedProof or 0x00000004;
	end_if;
	if drained then
		combinedProof := combinedProof or 0x00000008;
	end_if;

	if combinedProof <> LMC_OWNER_STARTUP_PROOF_REQUIRED then
		OwnershipStartupState[2]$UDINT := ObservationCycle;
		OwnershipStartupState[3] := 0;
		OwnershipStartupState[4]$UDINT := combinedProof;
		OwnershipStartupState[5]$UDINT := groupSignature;
		OwnershipStartupState[6]$UDINT := startupSnapshot[2];
		OwnershipStartupState[7]$UDINT := startupSnapshot[3];
		OwnershipStartupState[8]$UDINT := startupSnapshot[4];
		OwnershipStartupState[9]$UDINT := startupSnapshot[5];
		OwnershipStartupState[10]$UDINT := startupSnapshot[6];
		OwnershipStartupState[11]$UDINT := startupSnapshot[7];
		OwnershipStartupState[12]$UDINT := startupSnapshot[8];
		OwnershipStartupState[13]$UDINT := startupSnapshot[9];
		OwnershipStartupState[14] := 0;
		OwnershipStartupState[15] := 3;
		RETURN;
	end_if;

	signatureStable :=
		(OwnershipStartupState[4]$UDINT = combinedProof) &
		(OwnershipStartupState[5]$UDINT = groupSignature) &
		(OwnershipStartupState[6]$UDINT = startupSnapshot[2]) &
		(OwnershipStartupState[7]$UDINT = startupSnapshot[3]) &
		(OwnershipStartupState[8]$UDINT = startupSnapshot[4]) &
		(OwnershipStartupState[9]$UDINT = startupSnapshot[5]) &
		(OwnershipStartupState[10]$UDINT = startupSnapshot[6]) &
		(OwnershipStartupState[11]$UDINT = startupSnapshot[7]) &
		(OwnershipStartupState[12]$UDINT = startupSnapshot[8]) &
		(OwnershipStartupState[13]$UDINT = startupSnapshot[9]);

	freshObservation := FALSE;
	if OwnershipStartupState[3] <= 0 then
		OwnershipStartupState[3] := 1;
		OwnershipStartupState[14]$UDINT := ReportCycle;
		freshObservation := TRUE;
	elsif OwnershipStartupState[2]$UDINT <> ObservationCycle then
		freshObservation := TRUE;
		if signatureStable then
			if OwnershipStartupState[3] < LMC_OWNER_STARTUP_STABLE_SAMPLES then
				OwnershipStartupState[3] += 1;
			end_if;
		else
			OwnershipStartupState[3] := 1;
			OwnershipStartupState[14]$UDINT := ReportCycle;
		end_if;
	elsif signatureStable = FALSE then
		OwnershipStartupState[3] := 0;
		OwnershipStartupState[14] := 0;
		OwnershipStartupState[15] := 4;
	end_if;

	OwnershipStartupState[2]$UDINT := ObservationCycle;
	OwnershipStartupState[4]$UDINT := combinedProof;
	OwnershipStartupState[5]$UDINT := groupSignature;
	OwnershipStartupState[6]$UDINT := startupSnapshot[2];
	OwnershipStartupState[7]$UDINT := startupSnapshot[3];
	OwnershipStartupState[8]$UDINT := startupSnapshot[4];
	OwnershipStartupState[9]$UDINT := startupSnapshot[5];
	OwnershipStartupState[10]$UDINT := startupSnapshot[6];
	OwnershipStartupState[11]$UDINT := startupSnapshot[7];
	OwnershipStartupState[12]$UDINT := startupSnapshot[8];
	OwnershipStartupState[13]$UDINT := startupSnapshot[9];
	if OwnershipStartupState[3] > 0 then
		OwnershipStartupState[15] := 0;
	end_if;

	if OwnershipStartupState[3] < LMC_OWNER_STARTUP_STABLE_SAMPLES then
		RETURN;
	end_if;
	if freshObservation = FALSE then
		RETURN;
	end_if;
	stableElapsedMilliseconds := ReportCycle -
		OwnershipStartupState[14]$UDINT;
	if stableElapsedMilliseconds < LMC_OWNER_STARTUP_STABLE_MS then
		RETURN;
	end_if;

	_memset(dest:=#OwnershipState[0], usByte:=0, cntr:=1408);
	_memset(dest:=#OwnershipObserverState[0], usByte:=0, cntr:=432);
	_memset(dest:=#OwnershipLeaseState[0], usByte:=0,
		cntr:=sizeof(OwnershipLeaseState));
	_memset(dest:=#OwnershipPreemptedState[0], usByte:=0,
		cntr:=sizeof(OwnershipPreemptedState));
	_memset(dest:=#OwnershipIdentityState[0], usByte:=0,
		cntr:=sizeof(OwnershipIdentityState));
	_memset(dest:=#OwnershipLeaseIdentityState[0], usByte:=0,
		cntr:=sizeof(OwnershipLeaseIdentityState));
	_memset(dest:=#OwnershipPreemptedIdentityState[0], usByte:=0,
		cntr:=sizeof(OwnershipPreemptedIdentityState));
	OwnershipState[0]$UDINT := LMC_OWNER_TABLE_MAGIC;
	OwnershipState[3]$UDINT := DiagnosticsBootId;
	OwnershipState[4]$UDINT := ReportCycle;
	OwnershipState[5]$UDINT := LMC_OWNER_STARTUP_PROOF_REQUIRED;
	axisIndex := 1;
	while axisIndex <= LMC_OWNER_AXIS_COUNT do
		recordBase := LMC_OWNER_GLOBAL_SLOTS +
			((axisIndex - 1) * LMC_OWNER_AXIS_STRIDE);
		OwnershipState[recordBase] := axisIndex;
		OwnershipState[recordBase + 35]$UDINT :=
			LMC_OWNER_AXIS_RECORD_MAGIC + TO_UDINT(axisIndex);
		axisIndex += 1;
	end_while;
	Result := 0;

END_FUNCTION

FUNCTION GLOBAL LMCControlCommandService::NotifyAxisOwnershipSessionClosed
	VAR_INPUT
		SessionEpoch : UDINT;
	END_VAR
	VAR
		axisIndex : DINT;
		recordBase : DINT;
	END_VAR

	if SessionEpoch = 0 then
		RETURN;
	end_if;
	OwnershipState[22]$UDINT := SessionEpoch;
	axisIndex := 1;
	while axisIndex <= LMC_OWNER_AXIS_COUNT do
		recordBase := LMC_OWNER_GLOBAL_SLOTS +
			((axisIndex - 1) * LMC_OWNER_AXIS_STRIDE);
		if (OwnershipState[recordBase + 6]$UDINT = SessionEpoch) &
		   (OwnershipState[recordBase + 1] = LMC_OWNER_STATE_RESERVED) then
			OwnershipState[recordBase + 1] := LMC_OWNER_STATE_QUARANTINED;
			OwnershipState[recordBase + 32] :=
				LMC_OWNER_REPORT_QUARANTINE;
			OwnershipState[recordBase + 33] := -20;
		end_if;
		axisIndex += 1;
	end_while;

END_FUNCTION

FUNCTION GLOBAL LMCControlCommandService::ProcessAxisOwnership
	VAR
		latchSnapshot : ARRAY [0..303] OF USINT;
		startupSnapshot : ARRAY [0..11] OF UDINT;
		axisIndex : DINT;
		selectedAxisIndex : DINT;
		leaderAxisIndex : DINT;
		axisBit : UDINT;
		selectedAxisBit : UDINT;
		recordBase : DINT;
		selectedRecordBase : DINT;
		observerBase : DINT;
		selectedObserverBase : DINT;
		axisMask : UDINT;
		admissionToken : UDINT;
		ownerGeneration : UDINT;
		latchCycle : UDINT;
		serviceNow : UDINT;
		stableElapsed : UDINT;
		ownerElapsed : UDINT;
		commandId : DINT;
		ownerReference : DINT;
		ownerKind : DINT;
		ownerState : DINT;
		admissionMode : DINT;
		axisStatusRaw : UDINT;
		axisErrorRaw : UDINT;
		ds402StatusRaw : UDINT;
		profileErrorInfo : _LMCPROFERRORDEF;
		groupPowerState : DINT;
		groupLockState : DINT;
		groupFinished : DINT;
		groupError : DINT;
		latchCopyResult : DINT;
		startupCopyResult : DINT;
		publishResult : DINT;
		reportKind : UINT;
		allConnected : BOOL;
		allStandstill : BOOL;
		allPowerOn : BOOL;
		allPowerOff : BOOL;
		allErrorClear : BOOL;
		allTargetReached : BOOL;
		referencePowerOff : BOOL;
		powerOffEscalated : BOOL;
		tupleValid : BOOL;
		coherentObservation : BOOL;
		freshObservation : BOOL;
		terminalCandidate : BOOL;
		safeFailure : BOOL;
		forceQuarantine : BOOL;
		activitySeen : BOOL;
		unsupportedAxisSelected : BOOL;
	END_VAR

	if OwnershipState[0]$UDINT <> LMC_OWNER_TABLE_MAGIC then
		RETURN;
	end_if;
	OwnershipState[23]$UDINT := ops.tAbsolute;
	axisIndex := 1;
	while axisIndex <= LMC_OWNER_AXIS_COUNT do
		recordBase := LMC_OWNER_GLOBAL_SLOTS +
			((axisIndex - 1) * LMC_OWNER_AXIS_STRIDE);
		if OwnershipState[recordBase + 35]$UDINT <>
		   (LMC_OWNER_AXIS_RECORD_MAGIC + TO_UDINT(axisIndex)) then
			OwnershipState[24] := 1;
			OwnershipState[recordBase + 1] :=
				LMC_OWNER_STATE_QUARANTINED;
		end_if;
		axisIndex += 1;
	end_while;
	if LMC_AXIS_OWNERSHIP_ORDINARY_ENABLED = FALSE then
		RETURN;
	end_if;

	latchCopyResult := -1;
	startupCopyResult := -1;
	coherentObservation := FALSE;
	latchCycle := 0;
	if IsClientConnected(#InputLatch) then
		latchCopyResult := InputLatch.CopySnapshot(
			pDest:=#latchSnapshot[0], DestSize:=304);
		startupCopyResult := InputLatch.CopyAxisOwnershipStartupSnapshot(
			pDest:=#startupSnapshot[0], DestSize:=48);
	end_if;
	if (latchCopyResult = 0) & (startupCopyResult = 0) then
		latchCycle := latchSnapshot[0]$UDINT;
		coherentObservation :=
			(startupSnapshot[0] = LMC_OWNER_STARTUP_SNAPSHOT_MAGIC) &
			(latchCycle <> 0) & (startupSnapshot[1] = latchCycle) &
			((startupSnapshot[10] and
			  LMC_OWNER_LATCH_PHYSICAL_FLAG) <> 0) &
			(startupSnapshot[11] = 0) &
			(latchSnapshot[84]$UDINT = startupSnapshot[6]) &
			(latchSnapshot[120]$UDINT = startupSnapshot[7]) &
			(latchSnapshot[156]$UDINT = startupSnapshot[8]) &
			(latchSnapshot[192]$UDINT = startupSnapshot[9]);
	end_if;
	if coherentObservation = FALSE then
		latchCycle := 0;
	end_if;

	serviceNow := ops.tAbsolute;
	if serviceNow = 0 then
		serviceNow := 1;
	end_if;
	axisIndex := 1;
	while axisIndex <= LMC_OWNER_AXIS_COUNT do
		case axisIndex of
			1: axisBit := 0x00000001;
			2: axisBit := 0x00000002;
			3: axisBit := 0x00000004;
			4: axisBit := 0x00000008;
			5: axisBit := 0x00000010;
			6: axisBit := 0x00000020;
			7: axisBit := 0x00000040;
			8: axisBit := 0x00000080;
			9: axisBit := 0x00000100;
		else
			axisBit := 0;
		end_case;
		recordBase := LMC_OWNER_GLOBAL_SLOTS +
			((axisIndex - 1) * LMC_OWNER_AXIS_STRIDE);
		ownerState := OwnershipState[recordBase + 1];
		ownerKind := OwnershipState[recordBase + 2];
		if ((ownerKind = LMC_OWNER_KIND_DIRECT) |
		    (ownerKind = LMC_OWNER_KIND_GROUP)) &
		   ((ownerState = LMC_OWNER_STATE_DIRECT_ACTIVE) |
		    (ownerState = LMC_OWNER_STATE_GROUP_ACTIVE) |
		    (ownerState = LMC_OWNER_STATE_SAFETY_PREEMPTING)) then
			axisMask := OwnershipState[recordBase + 11]$UDINT;
			admissionToken := OwnershipState[recordBase + 4]$UDINT;
			ownerGeneration := OwnershipState[recordBase + 5]$UDINT;
			commandId := OwnershipState[recordBase + 3];
			ownerReference := OwnershipState[recordBase + 12];
			admissionMode := OwnershipState[recordBase + 14];
			leaderAxisIndex := 0;
			if (axisMask and 0x00000001) <> 0 then
				leaderAxisIndex := 1;
			elsif (axisMask and 0x00000002) <> 0 then
				leaderAxisIndex := 2;
			elsif (axisMask and 0x00000004) <> 0 then
				leaderAxisIndex := 3;
			elsif (axisMask and 0x00000008) <> 0 then
				leaderAxisIndex := 4;
			elsif (axisMask and 0x00000010) <> 0 then
				leaderAxisIndex := 5;
			elsif (axisMask and 0x00000020) <> 0 then
				leaderAxisIndex := 6;
			elsif (axisMask and 0x00000040) <> 0 then
				leaderAxisIndex := 7;
			elsif (axisMask and 0x00000080) <> 0 then
				leaderAxisIndex := 8;
			elsif (axisMask and 0x00000100) <> 0 then
				leaderAxisIndex := 9;
			end_if;

			if axisIndex = leaderAxisIndex then
				observerBase := (axisIndex - 1) * LMC_OWNER_OBSERVER_STRIDE;
				powerOffEscalated :=
					(OwnershipObserverState[observerBase + 5]$UDINT and
					 LMC_OWNER_OBSERVER_POWER_OFF_ESCALATED) <> 0;
				tupleValid := (axisMask <> 0) &
					(axisMask <= LMC_OWNER_ROBOT_AXIS_MASK) &
					(admissionToken <> 0) & (ownerGeneration <> 0);
				forceQuarantine := FALSE;
				unsupportedAxisSelected :=
					(axisMask and LMC_OWNER_UNSUPPORTED_AXIS_MASK) <> 0;
				selectedAxisIndex := 1;
				while selectedAxisIndex <= LMC_OWNER_AXIS_COUNT do
					case selectedAxisIndex of
						1: selectedAxisBit := 0x00000001;
						2: selectedAxisBit := 0x00000002;
						3: selectedAxisBit := 0x00000004;
						4: selectedAxisBit := 0x00000008;
						5: selectedAxisBit := 0x00000010;
						6: selectedAxisBit := 0x00000020;
						7: selectedAxisBit := 0x00000040;
						8: selectedAxisBit := 0x00000080;
						9: selectedAxisBit := 0x00000100;
					else
						selectedAxisBit := 0;
					end_case;
					selectedRecordBase := LMC_OWNER_GLOBAL_SLOTS +
						((selectedAxisIndex - 1) * LMC_OWNER_AXIS_STRIDE);
					selectedObserverBase :=
						(selectedAxisIndex - 1) * LMC_OWNER_OBSERVER_STRIDE;
					if (axisMask and selectedAxisBit) <> 0 then
						if (OwnershipState[selectedRecordBase + 1] <>
						    ownerState) |
						   (OwnershipState[selectedRecordBase + 2] <> ownerKind) |
						   (OwnershipState[selectedRecordBase + 3] <> commandId) |
						   (OwnershipState[selectedRecordBase + 4]$UDINT <>
						    admissionToken) |
						   (OwnershipState[selectedRecordBase + 5]$UDINT <>
						    ownerGeneration) |
						   (OwnershipState[selectedRecordBase + 11]$UDINT <>
						    axisMask) |
						   (OwnershipObserverState[selectedObserverBase]$UDINT <>
						    (LMC_OWNER_OBSERVER_MAGIC +
						     TO_UDINT(selectedAxisIndex))) |
						   (OwnershipObserverState[selectedObserverBase + 1]$UDINT <>
						    admissionToken) |
						   (OwnershipObserverState[selectedObserverBase + 2]$UDINT <>
						    ownerGeneration) |
						   (((OwnershipObserverState[selectedObserverBase + 5]$UDINT and
						      LMC_OWNER_OBSERVER_POWER_OFF_ESCALATED) <> 0) <>
						    powerOffEscalated) then
							tupleValid := FALSE;
						end_if;
						if (OwnershipObserverState[selectedObserverBase + 5]$UDINT and
						    LMC_OWNER_OBSERVER_FORCE_QUARANTINE) <> 0 then
							forceQuarantine := TRUE;
						end_if;
					end_if;
					selectedAxisIndex += 1;
				end_while;
				if powerOffEscalated &
				   (commandId <> LMC_OWNER_COMMAND_AXIS_STOP) &
				   (commandId <> LMC_OWNER_COMMAND_GROUP_DISABLE) &
				   (commandId <> LMC_OWNER_COMMAND_GROUP_STOP) then
					tupleValid := FALSE;
				end_if;
